           #C_E_Q_Unit := #C_E_Q_Unit + 1;
       ELSIF ((#E_Reactive_Rate1_Import < #MIN_ENERGY_VALUE) AND (#E_Reactive_Rate2_Import < #MIN_ENERGY_VALUE) AND
           (#E_Reactive_Rate1_Export < #MIN_ENERGY_VALUE) AND (#E_Reactive_Rate2_Export < #MIN_ENERGY_VALUE))
           AND (#C_E_Q_Unit > 1) THEN
           #C_E_Q_Unit := #C_E_Q_Unit - 1;
       ELSE
           ;
       END_IF;
       // selection apparent energy unit
       IF ((#E_Apparent_Rate1_Import > #MAX_ENERGY_VALUE) OR (#E_Apparent_Rate2_Import > #MAX_ENERGY_VALUE))
           AND (#C_E_S_Unit < 4) THEN
           #C_E_S_Unit := #C_E_S_Unit + 1;
       ELSIF ((#E_Apparent_Rate1_Import < #MIN_ENERGY_VALUE) AND (#E_Apparent_Rate2_Import < #MIN_ENERGY_VALUE))
           AND (#C_E_S_Unit > 1) THEN
           #C_E_S_Unit := #C_E_S_Unit - 1;
       ELSE
           ;
       END_IF;
   ELSE
       ;
   END_IF;
   //======================================================================================================================
   //==========calculate units=============================================================================================
   //======================================================================================================================    
   // calculate voltage unit
   CASE #C_U_Unit OF
       1:
           #U_Unit := 'mV';
           #U_L1_L2 := #ZU_L1_L2 * #THOUSAND;
           #U_L2_L3 := #ZU_L2_L3 * #THOUSAND;
           #U_L3_L1 := #ZU_L3_L1 * #THOUSAND;
           #U_L1 := #ZU_L1 * #THOUSAND;
           #U_L2 := #ZU_L2 * #THOUSAND;
           #U_L3 := #ZU_L3 * #THOUSAND;
           #U_L1_L2_min := #ZU_L1_L2_min * #THOUSAND;
           #U_L2_L3_min := #ZU_L2_L3_min * #THOUSAND;
           #U_L3_L1_min := #ZU_L3_L1_min * #THOUSAND;
           #U_L1_min := #ZU_L1_min * #THOUSAND;
           #U_L2_min := #ZU_L2_min * #THOUSAND;
           #U_L3_min := #ZU_L3_min * #THOUSAND;
           #U_L1_L2_max := #ZU_L1_L2_max * #THOUSAND;
           #U_L2_L3_max := #ZU_L2_L3_max * #THOUSAND;
           #U_L3_L1_max := #ZU_L3_L1_max * #THOUSAND;
           #U_L1_max := #ZU_L1_max * #THOUSAND;
           #U_L2_max := #ZU_L2_max * #THOUSAND;
           #U_L3_max := #ZU_L3_max * #THOUSAND;
           #U_PH_PH_Average := #ZU_PH_PH_Average * #THOUSAND;
           #U_PH_N_Average := #ZU_PH_N_Average * #THOUSAND;
           #U_PH_PH_Average_min := #ZU_PH_PH_Average_min * #THOUSAND;
           #U_PH_N_Average_min := #ZU_PH_N_Average_min * #THOUSAND;
           #U_PH_PH_Average_max := #ZU_PH_PH_Average_max * #THOUSAND;
           #U_PH_N_Average_max := #ZU_PH_N_Average_max * #THOUSAND;
       2:
           #U_Unit := 'V';
           #U_L1_L2 := #ZU_L1_L2;
           #U_L2_L3 := #ZU_L2_L3;
           #U_L3_L1 := #ZU_L3_L1;
           #U_L1 := #ZU_L1;
           #U_L2 := #ZU_L2;
           #U_L3 := #ZU_L3;
           #U_L1_L2_min := #ZU_L1_L2_min;
           #U_L2_L3_min := #ZU_L2_L3_min;
           #U_L3_L1_min := #ZU_L3_L1_min;
           #U_L1_min := #ZU_L1_min;
           #U_L2_min := #ZU_L2_min;
           #U_L3_min := #ZU_L3_min;
           #U_L1_L2_max := #ZU_L1_L2_max;
           #U_L2_L3_max := #ZU_L2_L3_max;
           #U_L3_L1_max := #ZU_L3_L1_max;
           #U_L1_max := #ZU_L1_max;
           #U_L2_max := #ZU_L2_max;
           #U_L3_max := #ZU_L3_max;
           #U_PH_PH_Average := #ZU_PH_PH_Average;
           #U_PH_N_Average := #ZU_PH_N_Average;
           #U_PH_PH_Average_min := #ZU_PH_PH_Average_min;
           #U_PH_N_Average_min := #ZU_PH_N_Average_min;
           #U_PH_PH_Average_max := #ZU_PH_PH_Average_max;
           #U_PH_N_Average_max := #ZU_PH_N_Average_max;
       ELSE:
           #U_Unit := 'kV';
           #U_L1_L2 := #ZU_L1_L2 / #THOUSAND;
           #U_L2_L3 := #ZU_L2_L3 / #THOUSAND;
           #U_L3_L1 := #ZU_L3_L1 / #THOUSAND;
           #U_L1 := #ZU_L1 / #THOUSAND;
           #U_L2 := #ZU_L2 / #THOUSAND;
           #U_L3 := #ZU_L3 / #THOUSAND;
           #U_L1_L2_min := #ZU_L1_L2_min / #THOUSAND;
           #U_L2_L3_min := #ZU_L2_L3_min / #THOUSAND;
           #U_L3_L1_min := #ZU_L3_L1_min / #THOUSAND;
           #U_L1_min := #ZU_L1_min / #THOUSAND;
           #U_L2_min := #ZU_L2_min / #THOUSAND;
           #U_L3_min := #ZU_L3_min / #THOUSAND;
           #U_L1_L2_max := #ZU_L1_L2_max / #THOUSAND;
           #U_L2_L3_max := #ZU_L2_L3_max / #THOUSAND;
           #U_L3_L1_max := #ZU_L3_L1_max / #THOUSAND;
           #U_L1_max := #ZU_L1_max / #THOUSAND;
           #U_L2_max := #ZU_L2_max / #THOUSAND;
           #U_L3_max := #ZU_L3_max / #THOUSAND;
           #U_PH_PH_Average := #ZU_PH_PH_Average / #THOUSAND;
           #U_PH_N_Average := #ZU_PH_N_Average / #THOUSAND;
           #U_PH_PH_Average_min := #ZU_PH_PH_Average_min / #THOUSAND;
           #U_PH_N_Average_min := #ZU_PH_N_Average_min / #THOUSAND;
           #U_PH_PH_Average_max := #ZU_PH_PH_Average_max / #THOUSAND;
           #U_PH_N_Average_max := #ZU_PH_N_Average_max / #THOUSAND;
   END_CASE;
   // calculate current unit    
   CASE #C_I_Unit OF
       1:
           #I_Unit := 'mA';
           #I_L1 := #ZI_L1 * #THOUSAND;
           #I_L2 := #ZI_L2 * #THOUSAND;
           #I_L3 := #ZI_L3 * #THOUSAND;
           #I_L1_min := #ZI_L1_min * #THOUSAND;
           #I_L2_min := #ZI_L2_min * #THOUSAND;
           #I_L3_min := #ZI_L3_min * #THOUSAND;
           #I_L1_max := #ZI_L1_max * #THOUSAND;
           #I_L2_max := #ZI_L2_max * #THOUSAND;
           #I_L3_max := #ZI_L3_max * #THOUSAND;
           #I_Average := #ZI_Average * #THOUSAND;
           #I_Average_min := #ZI_Average_min * #THOUSAND;
           #I_Average_max := #ZI_Average_max * #THOUSAND;
       2:
           #I_Unit := 'A';
           #I_L1 := #ZI_L1;
           #I_L2 := #ZI_L2;
           #I_L3 := #ZI_L3;
           #I_L1_min := #ZI_L1_min;
           #I_L2_min := #ZI_L2_min;
           #I_L3_min := #ZI_L3_min;
           #I_L1_max := #ZI_L1_max;
           #I_L2_max := #ZI_L2_max;
           #I_L3_max := #ZI_L3_max;
           #I_Average := #ZI_Average;
           #I_Average_min := #ZI_Average_min;
           #I_Average_max := #ZI_Average_max;
       ELSE:
           #I_Unit := 'kA';
           #I_L1 := #ZI_L1 / #THOUSAND;
           #I_L2 := #ZI_L2 / #THOUSAND;
           #I_L3 := #ZI_L3 / #THOUSAND;
           #I_L1_min := #ZI_L1_min / #THOUSAND;
           #I_L2_min := #ZI_L2_min / #THOUSAND;
           #I_L3_min := #ZI_L3_min / #THOUSAND;
           #I_L1_max := #ZI_L1_max / #THOUSAND;
           #I_L2_max := #ZI_L2_max / #THOUSAND;
           #I_L3_max := #ZI_L3_max / #THOUSAND;
           #I_Average := #ZI_Average / #THOUSAND;
           #I_Average_min := #ZI_Average_min / #THOUSAND;
           #I_Average_max := #ZI_Average_max / #THOUSAND;
   END_CASE;
   // calculate apparent power unit
   CASE #C_S_Unit OF
       1:
           #S_Unit := 'VA';
           #S_Total := #ZS_Total;
           #S_Total_min := #ZS_Total_min;
           #S_Total_max := #ZS_Total_max;
           #S_L1 := #ZS_L1;
           #S_L2 := #ZS_L2;
           #S_L3 := #ZS_L3;
           #S_L1_min := #ZS_L1_min;
           #S_L2_min := #ZS_L2_min;
           #S_L3_min := #ZS_L3_min;
           #S_L1_max := #ZS_L1_max;
           #S_L2_max := #ZS_L2_max;
           #S_L3_max := #ZS_L3_max;
       2:
           #S_Unit := 'kVA';
           #S_Total := #ZS_Total / #THOUSAND;
           #S_Total_min := #ZS_Total_min / #THOUSAND;
           #S_Total_max := #ZS_Total_max / #THOUSAND;
           #S_L1 := #ZS_L1 / #THOUSAND;
           #S_L2 := #ZS_L2 / #THOUSAND;
           #S_L3 := #ZS_L3 / #THOUSAND;
           #S_L1_min := #ZS_L1_min / #THOUSAND;
           #S_L2_min := #ZS_L2_min / #THOUSAND;
           #S_L3_min := #ZS_L3_min / #THOUSAND;
           #S_L1_max := #ZS_L1_max / #THOUSAND;
           #S_L2_max := #ZS_L2_max / #THOUSAND;
           #S_L3_max := #ZS_L3_max / #THOUSAND;
       3:
           #S_Unit := 'MVA';
           #S_Total := #ZS_Total / #MILLION;
           #S_Total_min := #ZS_Total_min / #MILLION;
           #S_Total_max := #ZS_Total_max / #MILLION;
           #S_L1 := #ZS_L1 / #MILLION;
           #S_L2 := #ZS_L2 / #MILLION;
           #S_L3 := #ZS_L3 / #MILLION;
           #S_L1_min := #ZS_L1_min / #MILLION;
           #S_L2_min := #ZS_L2_min / #MILLION;
           #S_L3_min := #ZS_L3_min / #MILLION;
           #S_L1_max := #ZS_L1_max / #MILLION;
           #S_L2_max := #ZS_L2_max / #MILLION;
           #S_L3_max := #ZS_L3_max / #MILLION;
       ELSE:
           #S_Unit := 'GVA';
           #S_Total := #ZS_Total / #MILLION / #THOUSAND;
           #S_Total_min := #ZS_Total_min / #MILLION / #THOUSAND;
           #S_Total_max := #ZS_Total_max / #MILLION / #THOUSAND;
           #S_L1 := #ZS_L1 / #MILLION / #THOUSAND;
           #S_L2 := #ZS_L2 / #MILLION / #THOUSAND;
           #S_L3 := #ZS_L3 / #MILLION / #THOUSAND;
           #S_L1_min := #ZS_L1_min / #MILLION / #THOUSAND;
           #S_L2_min := #ZS_L2_min / #MILLION / #THOUSAND;
           #S_L3_min := #ZS_L3_min / #MILLION / #THOUSAND;
           #S_L1_max := #ZS_L1_max / #MILLION / #THOUSAND;
           #S_L2_max := #ZS_L2_max / #MILLION / #THOUSAND;
           #S_L3_max := #ZS_L3_max / #MILLION / #THOUSAND;
   END_CASE;
   // calculate active power unit    
   CASE #C_P_Unit OF
       1:
           #P_Unit := 'W';
           #P_Total := #ZP_Total;
           #P_Total_min := #ZP_Total_min;
           #P_Total_max := #ZP_Total_max;
           #P_L1 := #ZP_L1;
           #P_L2 := #ZP_L2;
           #P_L3 := #ZP_L3;
           #P_L1_min := #ZP_L1_min;
           #P_L2_min := #ZP_L2_min;
           #P_L3_min := #ZP_L3_min;
           #P_L1_max := #ZP_L1_max;
           #P_L2_max := #ZP_L2_max;
           #P_L3_max := #ZP_L3_max;
       2:
           #P_Unit := 'kW';
           #P_Total := #ZP_Total / #THOUSAND;
           #P_Total_min := #ZP_Total_min / #THOUSAND;
           #P_Total_max := #ZP_Total_max / #THOUSAND;
           #P_L1 := #ZP_L1 / #THOUSAND;
           #P_L2 := #ZP_L2 / #THOUSAND;
           #P_L3 := #ZP_L3 / #THOUSAND;
           #P_L1_min := #ZP_L1_min / #THOUSAND;
           #P_L2_min := #ZP_L2_min / #THOUSAND;
           #P_L3_min := #ZP_L3_min / #THOUSAND;
           #P_L1_max := #ZP_L1_max / #THOUSAND;
           #P_L2_max := #ZP_L2_max / #THOUSAND;
           #P_L3_max := #ZP_L3_max / #THOUSAND;
       3:
           #P_Unit := 'MW';
           #P_Total := #ZP_Total / #MILLION;
           #P_Total_min := #ZP_Total_min / #MILLION;
           #P_Total_max := #ZP_Total_max / #MILLION;
           #P_L1 := #ZP_L1 / #MILLION;
           #P_L2 := #ZP_L2 / #MILLION;
           #P_L3 := #ZP_L3 / #MILLION;
           #P_L1_min := #ZP_L1_min / #MILLION;
           #P_L2_min := #ZP_L2_min / #MILLION;
           #P_L3_min := #ZP_L3_min / #MILLION;
           #P_L1_max := #ZP_L1_max / #MILLION;
           #P_L2_max := #ZP_L2_max / #MILLION;
           #P_L3_max := #ZP_L3_max / #MILLION;
       ELSE:
           #P_Unit := 'GW';
           #P_Total := #ZP_Total / #MILLION / #THOUSAND;
           #P_Total_min := #ZP_Total_min / #MILLION / #THOUSAND;
           #P_Total_max := #ZP_Total_max / #MILLION / #THOUSAND;
           #P_L1 := #ZP_L1 / #MILLION / #THOUSAND;
           #P_L2 := #ZP_L2 / #MILLION / #THOUSAND;
           #P_L3 := #ZP_L3 / #MILLION / #THOUSAND;
           #P_L1_min := #ZP_L1_min / #MILLION / #THOUSAND;
           #P_L2_min := #ZP_L2_min / #MILLION / #THOUSAND;
           #P_L3_min := #ZP_L3_min / #MILLION / #THOUSAND;
           #P_L1_max := #ZP_L1_max / #MILLION / #THOUSAND;
           #P_L2_max := #ZP_L2_max / #MILLION / #THOUSAND;
           #P_L3_max := #ZP_L3_max / #MILLION / #THOUSAND;
   END_CASE;
   // calculate reactive power unit   
   CASE #C_Q_Unit OF
       1:
           #Q_Unit := 'var';
           #Q_Total := #ZQ_Total;
           #Q_Total_min := #ZQ_Total_min;
           #Q_Total_max := #ZQ_Total_max;
           #Q_L1 := #ZQ_L1;
           #Q_L2 := #ZQ_L2;
           #Q_L3 := #ZQ_L3;
           #Q_L1_min := #ZQ_L1_min;
           #Q_L2_min := #ZQ_L2_min;
           #Q_L3_min := #ZQ_L3_min;
           #Q_L1_max := #ZQ_L1_max;
           #Q_L2_max := #ZQ_L2_max;
           #Q_L3_max := #ZQ_L3_max;
       2:
           #Q_Unit := 'kvar';
           #Q_Total := #ZQ_Total / #THOUSAND;
           #Q_Total_min := #ZQ_Total_min / #THOUSAND;
           #Q_Total_max := #ZQ_Total_max / #THOUSAND;
           #Q_L1 := #ZQ_L1 / #THOUSAND;
           #Q_L2 := #ZQ_L2 / #THOUSAND;
           #Q_L3 := #ZQ_L3 / #THOUSAND;
           #Q_L1_min := #ZQ_L1_min / #THOUSAND;
           #Q_L2_min := #ZQ_L2_min / #THOUSAND;
           #Q_L3_min := #ZQ_L3_min / #THOUSAND;
           #Q_L1_max := #ZQ_L1_max / #THOUSAND;
           #Q_L2_max := #ZQ_L2_max / #THOUSAND;
           #Q_L3_max := #ZQ_L3_max / #THOUSAND;
       3:
           #Q_Unit := 'Mvar';
           #Q_Total := #ZQ_Total / #MILLION;
           #Q_Total_min := #ZQ_Total_min / #MILLION;
           #Q_Total_max := #ZQ_Total_max / #MILLION;
           #Q_L1 := #ZQ_L1 / #MILLION;
           #Q_L2 := #ZQ_L2 / #MILLION;
           #Q_L3 := #ZQ_L3 / #MILLION;
           #Q_L1_min := #ZQ_L1_min / #MILLION;
           #Q_L2_min := #ZQ_L2_min / #MILLION;
           #Q_L3_min := #ZQ_L3_min / #MILLION;
           #Q_L1_max := #ZQ_L1_max / #MILLION;
           #Q_L2_max := #ZQ_L2_max / #MILLION;
           #Q_L3_max := #ZQ_L3_max / #MILLION;
       ELSE:
           #Q_Unit := 'Gvar';
           #Q_Total := #ZQ_Total / #MILLION / #THOUSAND;
           #Q_Total_min := #ZQ_Total_min / #MILLION / #THOUSAND;
           #Q_Total_max := #ZQ_Total_max / #MILLION / #THOUSAND;
           #Q_L1 := #ZQ_L1 / #MILLION / #THOUSAND;
           #Q_L2 := #ZQ_L2 / #MILLION / #THOUSAND;
           #Q_L3 := #ZQ_L3 / #MILLION / #THOUSAND;
           #Q_L1_min := #ZQ_L1_min / #MILLION / #THOUSAND;
           #Q_L2_min := #ZQ_L2_min / #MILLION / #THOUSAND;
           #Q_L3_min := #ZQ_L3_min / #MILLION / #THOUSAND;
           #Q_L1_max := #ZQ_L1_max / #MILLION / #THOUSAND;
           #Q_L2_max := #ZQ_L2_max / #MILLION / #THOUSAND;
           #Q_L3_max := #ZQ_L3_max / #MILLION / #THOUSAND;
   END_CASE;
   // calculate apparent energy unit     
   CASE #C_E_S_Unit OF
       1:
           IF ((#VEnergy_Meter_Unit[9] = TRUE) OR (#VEnergy_Meter_Unit[10] = TRUE)) THEN
               #S_Energy_Unit := 'kVAh';
               IF (#VEnergy_Meter_Unit[9] = FALSE) THEN
                   #E_Apparent_Rate1_Import := #ZE_Apparent_Rate1_Import / #THOUSAND;
               ELSE
                   #E_Apparent_Rate1_Import := #ZE_Apparent_Rate1_Import;
               END_IF;
               IF (#VEnergy_Meter_Unit[10] = FALSE) THEN
                   #E_Apparent_Rate2_Import := #ZE_Apparent_Rate2_Import / #THOUSAND;
               ELSE
                   #E_Apparent_Rate2_Import := #ZE_Apparent_Rate2_Import;
               END_IF;
           ELSE
               #S_Energy_Unit := 'VAh';
               #E_Apparent_Rate1_Import := #ZE_Apparent_Rate1_Import;
               #E_Apparent_Rate2_Import := #ZE_Apparent_Rate2_Import;
           END_IF;
       2:
           IF ((#VEnergy_Meter_Unit[9] = TRUE) OR (#VEnergy_Meter_Unit[10] = TRUE)) THEN
               #S_Energy_Unit := 'MVAh';
               IF (#VEnergy_Meter_Unit[9] = FALSE) THEN
                   #E_Apparent_Rate1_Import := #ZE_Apparent_Rate1_Import / #MILLION;
               ELSE
                   #E_Apparent_Rate1_Import := #ZE_Apparent_Rate1_Import / #THOUSAND;
               END_IF;
               IF (#VEnergy_Meter_Unit[10] = FALSE) THEN
                   #E_Apparent_Rate2_Import := #ZE_Apparent_Rate2_Import / #MILLION;
               ELSE
                   #E_Apparent_Rate2_Import := #ZE_Apparent_Rate2_Import / #THOUSAND;
               END_IF;
           ELSE
               #S_Energy_Unit := 'kVAh';
               #E_Apparent_Rate1_Import := #ZE_Apparent_Rate1_Import / #THOUSAND;
               #E_Apparent_Rate2_Import := #ZE_Apparent_Rate2_Import / #THOUSAND;
           END_IF;
       3:
           IF ((#VEnergy_Meter_Unit[9] = TRUE) OR (#VEnergy_Meter_Unit[10] = TRUE)) THEN
               #S_Energy_Unit := 'GVAh';
               IF (#VEnergy_Meter_Unit[9] = FALSE) THEN
                   #E_Apparent_Rate1_Import := #ZE_Apparent_Rate1_Import / #MILLION / #THOUSAND;
               ELSE
                   #E_Apparent_Rate1_Import := #ZE_Apparent_Rate1_Import / #MILLION;
               END_IF;
               IF (#VEnergy_Meter_Unit[10] = FALSE) THEN
                   #E_Apparent_Rate2_Import := #ZE_Apparent_Rate2_Import / #MILLION / #THOUSAND;
               ELSE
                   #E_Apparent_Rate2_Import := #ZE_Apparent_Rate2_Import / #MILLION;
               END_IF;
           ELSE
               #S_Energy_Unit := 'MVAh';
               #E_Apparent_Rate1_Import := #ZE_Apparent_Rate1_Import / #MILLION;
               #E_Apparent_Rate2_Import := #ZE_Apparent_Rate2_Import / #MILLION;
           END_IF;
       ELSE:
           IF ((#VEnergy_Meter_Unit[9] = TRUE) OR (#VEnergy_Meter_Unit[10] = TRUE)) THEN
               #S_Energy_Unit := 'TVAh';
               IF (#VEnergy_Meter_Unit[9] = FALSE) THEN
                   #E_Apparent_Rate1_Import := #ZE_Apparent_Rate1_Import / #MILLION / #MILLION;
               ELSE
                   #E_Apparent_Rate1_Import := #ZE_Apparent_Rate1_Import / #MILLION / #THOUSAND;
               END_IF;
               IF (#VEnergy_Meter_Unit[10] = FALSE) THEN
                   #E_Apparent_Rate2_Import := #ZE_Apparent_Rate2_Import / #MILLION / #MILLION;
               ELSE
                   #E_Apparent_Rate2_Import := #ZE_Apparent_Rate2_Import / #MILLION / #THOUSAND;
               END_IF;
           ELSE
               #S_Energy_Unit := 'GVAh';
               #E_Apparent_Rate1_Import := #ZE_Apparent_Rate1_Import / #MILLION / #THOUSAND;
               #E_Apparent_Rate2_Import := #ZE_Apparent_Rate2_Import / #MILLION / #THOUSAND;
           END_IF;
   END_CASE;
   // calculate active energy unit     
   CASE #C_E_P_Unit OF
       1:
           IF ((#VEnergy_Meter_Unit[1] = TRUE) OR (#VEnergy_Meter_Unit[2] = TRUE) OR
               (#VEnergy_Meter_Unit[3] = TRUE) OR (#VEnergy_Meter_Unit[4] = TRUE)) THEN
               #P_Energy_Unit := 'kWh';
               IF (#VEnergy_Meter_Unit[1] = FALSE) THEN
                   #E_Active_Rate1_Import := #ZE_Active_Rate1_Import / #THOUSAND;
               ELSE
                   #E_Active_Rate1_Import := #ZE_Active_Rate1_Import;
               END_IF;
               IF (#VEnergy_Meter_Unit[2] = FALSE) THEN
                   #E_Active_Rate2_Import := #ZE_Active_Rate2_Import / #THOUSAND;
               ELSE
                   #E_Active_Rate2_Import := #ZE_Active_Rate2_Import;
               END_IF;
               IF (#VEnergy_Meter_Unit[3] = FALSE) THEN
                   #E_Active_Rate1_Export := #ZE_Active_Rate1_Export / #THOUSAND;
               ELSE
                   #E_Active_Rate1_Export := #ZE_Active_Rate1_Export;
               END_IF;
               IF (#VEnergy_Meter_Unit[4] = FALSE) THEN
                   #E_Active_Rate1_Export := #ZE_Active_Rate1_Export / #THOUSAND;
               ELSE
                   #E_Active_Rate1_Export := #ZE_Active_Rate1_Export;
               END_IF;
           ELSE
               #P_Energy_Unit := 'Wh';
               #E_Active_Rate1_Import := #ZE_Active_Rate1_Import;
               #E_Active_Rate2_Import := #ZE_Active_Rate2_Import;
               #E_Active_Rate1_Export := #ZE_Active_Rate1_Export;
               #E_Active_Rate2_Export := #ZE_Active_Rate2_Export;
           END_IF;
       2:
           IF ((#VEnergy_Meter_Unit[1] = TRUE) OR (#VEnergy_Meter_Unit[2] = TRUE) OR
               (#VEnergy_Meter_Unit[3] = TRUE) OR (#VEnergy_Meter_Unit[4] = TRUE)) THEN
               #P_Energy_Unit := 'MWh';
               IF (#VEnergy_Meter_Unit[1] = FALSE) THEN
                   #E_Active_Rate1_Import := #ZE_Active_Rate1_Import / #MILLION;
               ELSE
                   #E_Active_Rate1_Import := #ZE_Active_Rate1_Import / #THOUSAND;
               END_IF;
               IF (#VEnergy_Meter_Unit[2] = FALSE) THEN
                   #E_Active_Rate2_Import := #ZE_Active_Rate2_Import / #MILLION;
               ELSE
                   #E_Active_Rate2_Import := #ZE_Active_Rate2_Import / #THOUSAND;
               END_IF;
               IF (#VEnergy_Meter_Unit[3] = FALSE) THEN
                   #E_Active_Rate1_Export := #ZE_Active_Rate1_Export / #MILLION;
               ELSE
                   #E_Active_Rate1_Export := #ZE_Active_Rate1_Export / #THOUSAND;
               END_IF;
               IF (#VEnergy_Meter_Unit[4] = FALSE) THEN
                   #E_Active_Rate2_Export := #ZE_Active_Rate2_Export / #MILLION;
               ELSE
                   #E_Active_Rate2_Export := #ZE_Active_Rate2_Export / #THOUSAND;
               END_IF;
           ELSE
               #P_Energy_Unit := 'kWh';
               #E_Active_Rate1_Import := #ZE_Active_Rate1_Import / #THOUSAND;
               #E_Active_Rate2_Import := #ZE_Active_Rate2_Import / #THOUSAND;
               #E_Active_Rate1_Export := #ZE_Active_Rate1_Export / #THOUSAND;
               #E_Active_Rate2_Export := #ZE_Active_Rate2_Export / #THOUSAND;
           END_IF;
       3:
           IF ((#VEnergy_Meter_Unit[1] = TRUE) OR (#VEnergy_Meter_Unit[2] = TRUE) OR
               (#VEnergy_Meter_Unit[3] = TRUE) OR (#VEnergy_Meter_Unit[4] = TRUE)) THEN
               #P_Energy_Unit := 'GWh';
               IF (#VEnergy_Meter_Unit[1] = FALSE) THEN
                   #E_Active_Rate1_Import := #ZE_Active_Rate1_Import / #MILLION / #THOUSAND;
               ELSE
                   #E_Active_Rate1_Import := #ZE_Active_Rate1_Import / #MILLION;
               END_IF;
               IF (#VEnergy_Meter_Unit[2] = FALSE) THEN
                   #E_Active_Rate2_Import := #ZE_Active_Rate2_Import / #MILLION / #THOUSAND;
               ELSE
                   #E_Active_Rate2_Import := #ZE_Active_Rate2_Import / #MILLION;
               END_IF;
               IF (#VEnergy_Meter_Unit[3] = FALSE) THEN
                   #E_Active_Rate1_Export := #ZE_Active_Rate1_Export / #MILLION / #THOUSAND;
               ELSE
                   #E_Active_Rate1_Export := #ZE_Active_Rate1_Export / #MILLION;
               END_IF;
               IF (#VEnergy_Meter_Unit[4] = FALSE) THEN
                   #E_Active_Rate2_Export := #ZE_Active_Rate2_Export / #MILLION / #THOUSAND;
               ELSE
                   #E_Active_Rate2_Export := #ZE_Active_Rate2_Export / #MILLION;
               END_IF;
           ELSE
               #P_Energy_Unit := 'MWh';
               #E_Active_Rate1_Import := #ZE_Active_Rate1_Import / #MILLION;
               #E_Active_Rate2_Import := #ZE_Active_Rate2_Import / #MILLION;
               #E_Active_Rate1_Export := #ZE_Active_Rate1_Export / #MILLION;
               #E_Active_Rate2_Export := #ZE_Active_Rate2_Export / #MILLION;
           END_IF;
       ELSE:
           IF ((#VEnergy_Meter_Unit[1] = TRUE) OR (#VEnergy_Meter_Unit[2] = TRUE) OR
               (#VEnergy_Meter_Unit[3] = TRUE) OR (#VEnergy_Meter_Unit[4] = TRUE)) THEN
               #P_Energy_Unit := 'TWh';
               IF (#VEnergy_Meter_Unit[1] = FALSE) THEN
                   #E_Active_Rate1_Import := #ZE_Active_Rate1_Import / #MILLION / #MILLION;
               ELSE
                   #E_Active_Rate1_Import := #ZE_Active_Rate1_Import / #MILLION / #THOUSAND;
               END_IF;
               IF (#VEnergy_Meter_Unit[2] = FALSE) THEN
                   #E_Active_Rate2_Import := #ZE_Active_Rate2_Import / #MILLION / #MILLION;
               ELSE
                   #E_Active_Rate2_Import := #ZE_Active_Rate2_Import / #MILLION / #THOUSAND;
               END_IF;
               IF (#VEnergy_Meter_Unit[3] = FALSE) THEN
                   #E_Active_Rate1_Export := #ZE_Active_Rate1_Export / #MILLION / #MILLION;
               ELSE
                   #E_Active_Rate1_Export := #ZE_Active_Rate1_Export / #MILLION / #THOUSAND;
               END_IF;
               IF (#VEnergy_Meter_Unit[4] = FALSE) THEN
                   #E_Active_Rate2_Export := #ZE_Active_Rate2_Export / #MILLION / #MILLION;
               ELSE
                   #E_Active_Rate2_Export := #ZE_Active_Rate2_Export / #MILLION / #THOUSAND;
               END_IF;
           ELSE
               #P_Energy_Unit := 'GWh';
               #E_Active_Rate1_Import := #ZE_Active_Rate1_Import / #MILLION / #THOUSAND;
               #E_Active_Rate2_Import := #ZE_Active_Rate2_Import / #MILLION / #THOUSAND;
               #E_Active_Rate1_Export := #ZE_Active_Rate1_Export / #MILLION / #THOUSAND;
               #E_Active_Rate2_Export := #ZE_Active_Rate2_Export / #MILLION / #THOUSAND;
           END_IF;
   END_CASE;
   // calculate reactive energy unit     
   CASE #C_E_Q_Unit OF
       1:
           IF ((#VEnergy_Meter_Unit[5] = TRUE) OR (#VEnergy_Meter_Unit[6] = TRUE) OR
               (#VEnergy_Meter_Unit[7] = TRUE) OR (#VEnergy_Meter_Unit[8] = TRUE)) THEN
               #Q_Energy_Unit := 'kWh';
               IF (#VEnergy_Meter_Unit[5] = FALSE) THEN
                   #E_Reactive_Rate1_Import := #ZE_Reactive_Rate1_Import / #THOUSAND;
               ELSE
                   #E_Reactive_Rate1_Import := #ZE_Reactive_Rate1_Import;
               END_IF;
               IF (#VEnergy_Meter_Unit[6] = FALSE) THEN
                   #E_Reactive_Rate2_Import := #ZE_Reactive_Rate2_Import / #THOUSAND;
               ELSE
                   #E_Reactive_Rate2_Import := #ZE_Reactive_Rate2_Import;
               END_IF;
               IF (#VEnergy_Meter_Unit[7] = FALSE) THEN
                   #E_Reactive_Rate1_Export := #ZE_Reactive_Rate1_Export / #THOUSAND;
               ELSE
                   #E_Reactive_Rate1_Export := #ZE_Reactive_Rate1_Export;
               END_IF;
               IF (#VEnergy_Meter_Unit[8] = FALSE) THEN
                   #E_Reactive_Rate2_Export := #ZE_Reactive_Rate2_Export / #THOUSAND;
               ELSE
                   #E_Reactive_Rate2_Export := #ZE_Reactive_Rate2_Export;
               END_IF;
           ELSE
               #Q_Energy_Unit := 'varh';
               #E_Reactive_Rate1_Import := #ZE_Reactive_Rate1_Import;
               #E_Reactive_Rate2_Import := #ZE_Reactive_Rate2_Import;
               #E_Reactive_Rate1_Export := #ZE_Reactive_Rate1_Export;
               #E_Reactive_Rate2_Export := #ZE_Reactive_Rate2_Export;
           END_IF;
       2:
           IF ((#VEnergy_Meter_Unit[5] = TRUE) OR (#VEnergy_Meter_Unit[6] = TRUE) OR
               (#VEnergy_Meter_Unit[7] = TRUE) OR (#VEnergy_Meter_Unit[8] = TRUE)) THEN
               #Q_Energy_Unit := 'MWh';
               IF (#VEnergy_Meter_Unit[5] = FALSE) THEN
                   #E_Reactive_Rate1_Import := #ZE_Reactive_Rate1_Import / #MILLION;
               ELSE
                   #E_Reactive_Rate1_Import := #ZE_Reactive_Rate1_Import;
               END_IF;
               IF (#VEnergy_Meter_Unit[6] = FALSE) THEN
                   #E_Reactive_Rate2_Import := #ZE_Reactive_Rate2_Import / #MILLION;
               ELSE
                   #E_Reactive_Rate2_Import := #ZE_Reactive_Rate2_Import;
               END_IF;
               IF (#VEnergy_Meter_Unit[7] = FALSE) THEN
                   #E_Reactive_Rate1_Export := #ZE_Reactive_Rate1_Export / #MILLION;
               ELSE
                   #E_Reactive_Rate1_Export := #ZE_Reactive_Rate1_Export;
               END_IF;
               IF (#VEnergy_Meter_Unit[8] = FALSE) THEN
                   #E_Reactive_Rate2_Export := #ZE_Reactive_Rate2_Export / #MILLION;
               ELSE
                   #E_Reactive_Rate2_Export := #ZE_Reactive_Rate2_Export;
               END_IF;
           ELSE
               #Q_Energy_Unit := 'kvarh';
               #E_Reactive_Rate1_Import := #ZE_Reactive_Rate1_Import / #THOUSAND;
               #E_Reactive_Rate2_Import := #ZE_Reactive_Rate2_Import / #THOUSAND;
               #E_Reactive_Rate1_Export := #ZE_Reactive_Rate1_Export / #THOUSAND;
               #E_Reactive_Rate2_Export := #ZE_Reactive_Rate2_Export / #THOUSAND;
           END_IF;
       3:
           IF ((#VEnergy_Meter_Unit[5] = TRUE) OR (#VEnergy_Meter_Unit[6] = TRUE) OR
               (#VEnergy_Meter_Unit[7] = TRUE) OR (#VEnergy_Meter_Unit[8] = TRUE)) THEN
               #Q_Energy_Unit := 'GWh';
               IF (#VEnergy_Meter_Unit[5] = FALSE) THEN
                   #E_Reactive_Rate1_Import := #ZE_Reactive_Rate1_Import / #MILLION / #THOUSAND;
               ELSE
                   #E_Reactive_Rate1_Import := #ZE_Reactive_Rate1_Import / #THOUSAND;
               END_IF;
               IF (#VEnergy_Meter_Unit[6] = FALSE) THEN
                   #E_Reactive_Rate2_Import := #ZE_Reactive_Rate2_Import / #MILLION / #THOUSAND;
               ELSE
                   #E_Reactive_Rate2_Import := #ZE_Reactive_Rate2_Import / #THOUSAND;
               END_IF;
               IF (#VEnergy_Meter_Unit[7] = FALSE) THEN
                   #E_Reactive_Rate1_Export := #ZE_Reactive_Rate1_Export / #MILLION / #THOUSAND;
               ELSE
                   #E_Reactive_Rate1_Export := #ZE_Reactive_Rate1_Export / #THOUSAND;
               END_IF;
               IF (#VEnergy_Meter_Unit[8] = FALSE) THEN
                   #E_Reactive_Rate2_Export := #ZE_Reactive_Rate2_Export / #MILLION / #THOUSAND;
               ELSE
                   #E_Reactive_Rate2_Export := #ZE_Reactive_Rate2_Export / #THOUSAND;
               END_IF;
           ELSE
               #Q_Energy_Unit := 'Mvarh';
               #E_Reactive_Rate1_Import := #ZE_Reactive_Rate1_Import / #MILLION;
               #E_Reactive_Rate2_Import := #ZE_Reactive_Rate2_Import / #MILLION;
               #E_Reactive_Rate1_Export := #ZE_Reactive_Rate1_Export / #MILLION;
               #E_Reactive_Rate2_Export := #ZE_Reactive_Rate2_Export / #MILLION;
           END_IF;
       ELSE:
           IF ((#VEnergy_Meter_Unit[5] = TRUE) OR (#VEnergy_Meter_Unit[6] = TRUE) OR
               (#VEnergy_Meter_Unit[7] = TRUE) OR (#VEnergy_Meter_Unit[8] = TRUE)) THEN
               #Q_Energy_Unit := 'TWh';
               IF (#VEnergy_Meter_Unit[5] = FALSE) THEN
                   #E_Reactive_Rate1_Import := #ZE_Reactive_Rate1_Import / #MILLION / #MILLION;
               ELSE
                   #E_Reactive_Rate1_Import := #ZE_Reactive_Rate1_Import / #MILLION / #THOUSAND;
               END_IF;
               IF (#VEnergy_Meter_Unit[6] = FALSE) THEN
                   #E_Reactive_Rate2_Import := #ZE_Reactive_Rate2_Import / #MILLION / #MILLION;
               ELSE
                   #E_Reactive_Rate2_Import := #ZE_Reactive_Rate2_Import / #MILLION / #THOUSAND;
               END_IF;
               IF (#VEnergy_Meter_Unit[7] = FALSE) THEN
                   #E_Reactive_Rate1_Export := #ZE_Reactive_Rate1_Export / #MILLION / #MILLION;
               ELSE
                   #E_Reactive_Rate1_Export := #ZE_Reactive_Rate1_Export / #MILLION / #THOUSAND;
               END_IF;
               IF (#VEnergy_Meter_Unit[8] = FALSE) THEN
                   #E_Reactive_Rate2_Export := #ZE_Reactive_Rate2_Export / #MILLION / #MILLION;
               ELSE
                   #E_Reactive_Rate2_Export := #ZE_Reactive_Rate2_Export / #MILLION / #THOUSAND;
               END_IF;
           ELSE
               #Q_Energy_Unit := 'Gvarh';
               #E_Reactive_Rate1_Import := #ZE_Reactive_Rate1_Import / #MILLION / #THOUSAND;
               #E_Reactive_Rate2_Import := #ZE_Reactive_Rate2_Import / #MILLION / #THOUSAND;
               #E_Reactive_Rate1_Export := #ZE_Reactive_Rate1_Export / #MILLION / #THOUSAND;
               #E_Reactive_Rate2_Export := #ZE_Reactive_Rate2_Export / #MILLION / #THOUSAND;
           END_IF;
   END_CASE;
   //======================================================================================================================
   //==========calculate scale final value=================================================================================
   //======================================================================================================================        
   // calculate scale final voltage PH-PH
   IF ((#AREA_TO_THOUSAND < #U_L1_L2_max) OR (#AREA_TO_THOUSAND < #U_L2_L3_max) OR (#AREA_TO_THOUSAND < #U_L3_L1_max)) THEN
       #ZScale_End_U_PH_PH := #ZSCALE_END_I4;
   ELSIF ((#AREA_TO_HUNDRED < #U_L1_L2_max) OR (#AREA_TO_HUNDRED < #U_L2_L3_max) OR (#AREA_TO_HUNDRED < #U_L3_L1_max)) THEN
       #ZScale_End_U_PH_PH := #ZSCALE_END_I3;
   ELSIF ((#AREA_TO_TEN < #U_L1_L2_max) OR (#AREA_TO_TEN < #U_L2_L3_max) OR (#AREA_TO_TEN < #U_L3_L1_max)) THEN
       #ZScale_End_U_PH_PH := #ZSCALE_END_I2;
   ELSIF ((0 <= #U_L1_L2_max) OR (0 <= #U_L2_L3_max) OR (0 <= #U_L3_L1_max)) THEN
       #ZScale_End_U_PH_PH := #ZSCALE_END_I1;
   ELSE
       ;
   END_IF;
   // selection maximum value
   #U_PH_PH := MAX(IN1 := #U_L1_L2_max, IN2 := #U_L2_L3_max, IN3 := #U_L3_L1_max, IN4 := 4.0);
   // 
   #Scale_End_U_PH_PH := (REAL_TO_DINT(#U_PH_PH * #FACTOR)) + (#ZScale_End_U_PH_PH - (REAL_TO_DINT(#U_PH_PH * #FACTOR) MOD #ZScale_End_U_PH_PH));
   // calculate scale final voltage PH-N
   IF ((#AREA_TO_THOUSAND < #U_L1_max) OR (#AREA_TO_THOUSAND < #U_L2_max) OR (#AREA_TO_THOUSAND < #U_L3_max)) THEN
       #ZScale_End_U_PH_N := #ZSCALE_END_I4;
   ELSIF ((#AREA_TO_HUNDRED < #U_L1_max) OR (#AREA_TO_HUNDRED < #U_L2_max) OR (#AREA_TO_HUNDRED < #U_L3_max)) THEN
       #ZScale_End_U_PH_N := #ZSCALE_END_I3;
   ELSIF ((#AREA_TO_TEN < #U_L1_max) OR (#AREA_TO_TEN < #U_L2_max) OR (#AREA_TO_TEN < #U_L3_max)) THEN
       #ZScale_End_U_PH_N := #ZSCALE_END_I2;
   ELSIF ((0 <= #U_L1_max) OR (0 <= #U_L2_max) OR (0 <= #U_L3_max)) THEN
       #ZScale_End_U_PH_N := #ZSCALE_END_I1;
   ELSE
       ;
   END_IF;
   // selection maximum value
   #U_PH_N := MAX(IN1 := #U_L1_max, IN2 := #U_L2_max, IN3 := #U_L3_max, IN4 := 4.0);
   // 
   #Scale_End_U_PH_N := (REAL_TO_DINT(#U_PH_N * #FACTOR)) + (#ZScale_End_U_PH_N - (REAL_TO_DINT(#U_PH_N * #FACTOR) MOD #ZScale_End_U_PH_N));
   // calculate scale final current
   IF ((#AREA_TO_THOUSAND < #I_L1_max) OR (#AREA_TO_THOUSAND < #I_L2_max) OR (#AREA_TO_THOUSAND < #I_L3_max)) THEN
       #ZScale_End_I := #ZSCALE_END_I4;
   ELSIF ((#AREA_TO_HUNDRED < #I_L1_max) OR (#AREA_TO_HUNDRED < #I_L2_max) OR (#AREA_TO_HUNDRED < #I_L3_max)) THEN
       #ZScale_End_I := #ZSCALE_END_I3;
   ELSIF ((#AREA_TO_TEN < #I_L1_max) OR (#AREA_TO_TEN < #I_L2_max) OR (#AREA_TO_TEN < #I_L3_max)) THEN
       #ZScale_End_I := #ZSCALE_END_I2;
   ELSIF ((0 <= #I_L1_max) OR (0 <= #I_L2_max) OR (0 <= #I_L3_max)) THEN
       #ZScale_End_I := #ZSCALE_END_I1;
   ELSE
       ;
   END_IF;
   // selection maximum value
   #I := MAX(IN1 := #I_L1_max, IN2 := #I_L2_max, IN3 := #I_L3_max, IN4 := 4.0);
   //
   #Scale_End_I := (REAL_TO_DINT(#I * #FACTOR)) + (#ZScale_End_I - (REAL_TO_DINT(#I * #FACTOR) MOD #ZScale_End_I));
   // calculate scale final apparent power    
   IF ((#AREA_TO_THOUSAND < #S_L1_max) OR (#AREA_TO_THOUSAND < #S_L2_max) OR
       (#AREA_TO_THOUSAND < #S_L3_max) OR (#AREA_TO_THOUSAND < #S_Total_max)) THEN
       #ZScale_End_S := #ZSCALE_END_SPQ4;
   ELSIF ((#AREA_TO_HUNDRED < #S_L1_max) OR (#AREA_TO_HUNDRED < #S_L2_max) OR
       (#AREA_TO_HUNDRED < #S_L3_max) OR (#AREA_TO_HUNDRED < #S_Total_max)) THEN
       #ZScale_End_S := #ZSCALE_END_SPQ3;
   ELSIF ((#AREA_TO_TEN < #S_L1_max) OR (#AREA_TO_TEN < #S_L2_max) OR
       (#AREA_TO_TEN < #S_L3_max) OR (#AREA_TO_TEN < #S_Total_max)) THEN
       #ZScale_End_S := #ZSCALE_END_SPQ2;
   ELSIF ((0 <= #S_L1_max) OR (0 <= #S_L2_max) OR (0 <= #S_L3_max) OR (0 <= #S_Total_max)) THEN
       #ZScale_End_S := #ZSCALE_END_SPQ1;
   ELSE
       ;
   END_IF;
   // selection maximum value 
   #S := MAX(IN1 := #S_L1_max, IN2 := #S_L2_max, IN3 := #S_L3_max, IN4 := #S_Total_max, IN5 := 4.0);
   //
   #Scale_End_S := (REAL_TO_DINT(#S * #FACTOR)) + (#ZScale_End_S - (REAL_TO_DINT(#S * #FACTOR) MOD #ZScale_End_S));
   // calculate scale final active power
   IF ((#AREA_TO_THOUSAND < #P_L1_max) OR (#AREA_TO_THOUSAND < #P_L2_max) OR
       (#AREA_TO_THOUSAND < #P_L3_max) OR (#AREA_TO_THOUSAND < #P_Total_max)) THEN
       #ZScale_End_P := #ZSCALE_END_SPQ4;
   ELSIF ((#AREA_TO_HUNDRED < #P_L1_max) OR (#AREA_TO_HUNDRED < #P_L2_max) OR
       (#AREA_TO_HUNDRED < #P_L3_max) OR (#AREA_TO_HUNDRED < #P_Total_max)) THEN
       #ZScale_End_P := #ZSCALE_END_SPQ3;
   ELSIF ((#AREA_TO_TEN < #P_L1_max) OR (#AREA_TO_TEN < #P_L2_max) OR
       (#AREA_TO_TEN < #P_L3_max) OR (#AREA_TO_TEN < #P_Total_max)) THEN
       #ZScale_End_P := #ZSCALE_END_SPQ2;
   ELSIF ((0 <= #P_L1_max) OR (0 <= #P_L2_max) OR (0 <= #P_L3_max) OR (0 <= #P_Total_max)) THEN
       #ZScale_End_P := #ZSCALE_END_SPQ1;
   ELSE
       ;
   END_IF;
   // selection maximum value
   #P := MAX(IN1 := #P_L1_max, IN2 := #P_L2_max, IN3 := #P_L3_max, IN4 := #P_Total_max, IN5 := 4.0);
   //
   #Scale_End_P := (REAL_TO_DINT(#P * #FACTOR)) + (#ZScale_End_P - (REAL_TO_DINT(#P * #FACTOR) MOD #ZScale_End_P));
   // calculate scale final reactive power max
   IF ((#AREA_TO_THOUSAND < #Q_L1_max) OR (#AREA_TO_THOUSAND < #Q_L2_max) OR
       (#AREA_TO_THOUSAND < #Q_L3_max) OR (#AREA_TO_THOUSAND < #Q_Total_max) OR
       (- #AREA_TO_THOUSAND > #Q_L1_min) OR (- #AREA_TO_THOUSAND > #Q_L2_min) OR
       (- #AREA_TO_THOUSAND > #Q_L3_min) OR (- #AREA_TO_THOUSAND > #Q_Total_min)) THEN
       #ZScale_End_Q := #ZSCALE_END_SPQ4;
   ELSIF ((#AREA_TO_HUNDRED < #Q_L1_max) OR (#AREA_TO_HUNDRED < #Q_L2_max) OR
       (#AREA_TO_HUNDRED < #Q_L3_max) OR (#AREA_TO_HUNDRED < #Q_Total_max) OR
       (- #AREA_TO_HUNDRED > #Q_L1_min) OR (- #AREA_TO_HUNDRED > #Q_L2_min) OR
       (- #AREA_TO_HUNDRED > #Q_L3_min) OR (- #AREA_TO_HUNDRED > #Q_Total_min)) THEN
       #ZScale_End_Q := #ZSCALE_END_SPQ3;
   ELSIF ((#AREA_TO_TEN < #Q_L1_max) OR (#AREA_TO_TEN < #Q_L2_max) OR
       (#AREA_TO_TEN < #Q_L3_max) OR (#AREA_TO_TEN < #Q_Total_max) OR
       (- #AREA_TO_TEN > #Q_L1_min) OR (- #AREA_TO_TEN > #Q_L2_min) OR
       (- #AREA_TO_TEN > #Q_L3_min) OR (- #AREA_TO_TEN > #Q_Total_min)) THEN
       #ZScale_End_Q := #ZSCALE_END_SPQ2;
   ELSIF ((0 <= #Q_L1_max) OR (0 <= #Q_L2_max) OR (0 <= #Q_L3_max) OR (0 <= #Q_Total_max) OR
       (0 >= #Q_L1_min) OR (0 >= #Q_L2_min) OR (0 >= #Q_L3_min) OR (0 >= #Q_Total_min)) THEN
       #ZScale_End_Q := #ZSCALE_END_SPQ1;
   ELSE
       ;
   END_IF;
   // calculate scale final reactive power max
   IF ((MAX(IN1 := #Q_L1_max, IN2 := #Q_L2_max, IN3 := #Q_L3_max, IN4 := #Q_Total_max)) = 0) THEN
       #Q := 4.0;
   ELSE
       #Q := MAX(IN1 := #Q_L1_max, IN2 := #Q_L2_max, IN3 := #Q_L3_max, IN4 := #Q_Total_max);
   END_IF;
   //
   IF (#Q > 0) THEN
       #Scale_End_Q := (REAL_TO_DINT(#Q * #FACTOR)) + (#ZScale_End_Q - (REAL_TO_DINT(#Q * #FACTOR) MOD #ZScale_End_Q));
   ELSIF (#Q < 0) THEN
       #Scale_End_Q := (REAL_TO_DINT(#Q * #FACTOR)) - (#ZScale_End_Q - (REAL_TO_DINT(#Q * #FACTOR) MOD #ZScale_End_Q));
   ELSE
       ;
   END_IF;
   // calculate scale final reactive power min
   IF ((MIN(IN1 := #Q_L1_min, IN2 := #Q_L2_min, IN3 := #Q_L3_min, IN4 := #Q_Total_min)) = 0) THEN
       #Q_min := -4.0;
   ELSE
       #Q_min := MIN(IN1 := #Q_L1_min, IN2 := #Q_L2_min, IN3 := #Q_L3_min, IN4 := #Q_Total_min);
   END_IF;
   //
   IF (#Q_min > 0) THEN
       #Scale_Begin_Q := 0;
   ELSIF (#Q_min < 0) THEN
       #Scale_Begin_Q := (REAL_TO_DINT(#Q_min * #FACTOR)) - (#ZScale_End_Q - (REAL_TO_DINT(#Q_min * #FACTOR) MOD #ZScale_End_Q));
   END_IF;
   //======================================================================================================================
   //==========value to output value=======================================================================================
   //======================================================================================================================
   // calculation value
   #Calculate_Value1 := #Driver_Data.Calculate_Value1;               // calculate value 1
   #Calculate_Value2 := #Driver_Data.Calculate_Value2;               // calculate value 2
   #Calculate_Value3 := #Driver_Data.Calculate_Value3;               // calculate value 3
   #Calculate_Value4 := #Driver_Data.Calculate_Value4;               // calculate value 4
   #Calculate_Value5 := #Driver_Data.Calculate_Value5;               // calculate value 5
   #Calculate_Value6 := #Driver_Data.Calculate_Value6;               // calculate value 6
   // selection of show modification
   #U_PH_PH_Mod := #Driver_Data.U_PH_PH_Mod;                    // voltage PH-PH show modification
   #U_PH_N_Mod := #Driver_Data.U_PH_N_Mod;                     // voltage PH-N show modification
   #I_Mod := #Driver_Data.I_Mod;                          // current show modification
   #S_Mod := #Driver_Data.S_Mod;                          // apparent power show modification
   #P_Mod := #Driver_Data.P_Mod;                          // active power show modification
   #Q_Mod := #Driver_Data.Q_Mod;                          // reactive power show modification
   #E_Mod := #Driver_Data.E_Mod;                          // energy meter show modification
   #f_Mod := #Driver_Data.f_Mod;                          // frequenz show modification
   #Cos_Mod := #Driver_Data.Cos_Mod;                        // efficiency factor show modification  
   // temp value to output value
   #f := #Zf;                                         // frequency
   #f_min := #Zf_min;                                     // minimum frequenz
   #f_max := #Zf_max;                                     // maximum frequenz
   #Cos_Total := #ZCos_Total;                                 // total efficiency factor
   #Cos_Total_min := #ZCos_Total_min;                             // minimum total efficiency factor
   #Cos_Total_max := #ZCos_Total_max;                             // maximum total efficiency factor
   #Cos_L1 := #ZCos_L1;                                    // efficiency factor L1       
   #Cos_L1_min := #ZCos_L1_min;                                // minimum efficiency factor L1
   #Cos_L1_max := #ZCos_L1_max;                                // maximum efficiency factor L1
   #Cos_L2 := #ZCos_L2;                                    // efficiency factor L2
   #Cos_L2_min := #ZCos_L2_min;                                // minimum efficiency factor L2
   #Cos_L2_max := #ZCos_L2_max;                                // maximum efficiency factor L2
   #Cos_L3 := #ZCOS_L3;                                    // efficiency factor L3
   #Cos_L3_min := #ZCos_L3_min;                                // minimum efficiency factor L3
   #Cos_L3_max := #ZCos_L3_max;                                // maximum efficiency factor L3
   // reset time Energy  
   #RTime_Data_Energy := #Driver_Data.RTime_Data_Energy;              // Reset Time
   #R_Year_Energy := BCD16_TO_INT(#ZRTime_Data_Energy[1]) + 100;      // Reset year   
   #R_Month_Energy := BCD16_TO_INT(#ZRTime_Data_Energy[2]) + 100;      // Reset month
   #R_Day_Energy := BCD16_TO_INT(#ZRTime_Data_Energy[3]) + 100;      // Reset day    
   #R_Hour_Energy := BCD16_TO_INT(#ZRTime_Data_Energy[4]) + 100;      // Reset hour   
   #R_Minute_Energy := BCD16_TO_INT(#ZRTime_Data_Energy[5]) + 100;      // Reset minute 
   #R_Second_Energy := BCD16_TO_INT(#ZRTime_Data_Energy[6]) + 100;      // Reset Second
   // reset time value
   #RTime_Data_Value := #Driver_Data.RTime_Data_Value;               // Reset Time
   #R_Year_Value := BCD16_TO_INT(#ZRTime_Data_Value[1]) + 100;       // Reset year   
   #R_Month_Value := BCD16_TO_INT(#ZRTime_Data_Value[2]) + 100;       // Reset month  
   #R_Day_Value := BCD16_TO_INT(#ZRTime_Data_Value[3]) + 100;       // Reset day    
   #R_Hour_Value := BCD16_TO_INT(#ZRTime_Data_Value[4]) + 100;       // Reset hour   
   #R_Minute_Value := BCD16_TO_INT(#ZRTime_Data_Value[5]) + 100;       // Reset minute 
   #R_Second_Value := BCD16_TO_INT(#ZRTime_Data_Value[6]) + 100;       // Reset Second
   // HMI_Bits
   IF (#Driver_Data.Rest_Start_Auto = TRUE) THEN
       #Start_Auto := FALSE;
       #Start_Acyclic := FALSE;
   ELSE
       ;
   END_IF;
   #HMI_Bits.Start_Acyclic := #Start_Acyclic;
   #HMI_Bits.Start_Auto := #Start_Auto;
   #HMI_Bits.Reset_min_max_Data := #Reset_min_max_Data;
   #HMI_Bits.Reset_Energy_Meter := #Reset_Energy_Meter;
   //
   #Read_Value := #Driver_Data.Read_Value;
   //======================================================================================================================
   //==========error code==================================================================================================
   //======================================================================================================================  
   // error code output
   #ERROR := #Fehler;
END_FUNCTION_BLOCK

FUNCTION_BLOCK "LAnInput6Lim"   // FB1750, FBD
TITLE = LAnInput6Lim
{ S7_Optimized_Access := 'FALSE' }
AUTHOR : VCC
FAMILY : ProcEqp
NAME : AnInput
VERSION : 1.0
// ================================================================================
// This module is used to read an analogue Input value and scale it. 
// It also gives the possibility to define 6 limits (High High High, High High, 
// High, Low, Low Low and Low Low Low level) and to create 6 alarms for these 
// limits. 
// ================================================================================
// stored: AutoNumber false, IsIECCheckEnabled false, SetENOAutomatically False, UDAEnableTagReadback false
   VAR_INPUT
      I_AnInput { ExternalAccessible := 'False'; ExternalVisible := 'False'; ExternalWritable := 'False'} : Real;   // Analogue Input Value
      I_MotorActive { ExternalAccessible := 'False'; ExternalVisible := 'False'; ExternalWritable := 'False'} : Bool;
      I_EnHHHAlarm { ExternalAccessible := 'False'; ExternalVisible := 'False'; ExternalWritable := 'False'} : Bool;   // Enable HHH Limit Alarm
      I_ResHHHAlarm { ExternalAccessible := 'False'; ExternalVisible := 'False'; ExternalWritable := 'False'} : Bool;   // Reset HHH Limit Alarm
      I_EnHHAlarm { ExternalAccessible := 'False'; ExternalVisible := 'False'; ExternalWritable := 'False'} : Bool;   // Enable HH Limit Alarm
      I_ResHHAlarm { ExternalAccessible := 'False'; ExternalVisible := 'False'; ExternalWritable := 'False'} : Bool;   // Reset HH Limit Alarm
      I_EnHAlarm { ExternalAccessible := 'False'; ExternalVisible := 'False'; ExternalWritable := 'False'} : Bool;   // Enable H Limit Alarm
      I_ResHAlarm { ExternalAccessible := 'False'; ExternalVisible := 'False'; ExternalWritable := 'False'} : Bool;   // Reset H Limit Alarm
      I_EnLAlarm { ExternalAccessible := 'False'; ExternalVisible := 'False'; ExternalWritable := 'False'} : Bool;   // Enable L Limit Alarm
      I_ResLAlarm { ExternalAccessible := 'False'; ExternalVisible := 'False'; ExternalWritable := 'False'} : Bool;   // Reset L Limit Alarm
      I_EnLLAlarm { ExternalAccessible := 'False'; ExternalVisible := 'False'; ExternalWritable := 'False'} : Bool;   // Enable LL Limit Alarm
      I_ResLLAlarm { ExternalAccessible := 'False'; ExternalVisible := 'False'; ExternalWritable := 'False'} : Bool;   // Reset LL Limit Alarm
      I_EnLLLAlarm { ExternalAccessible := 'False'; ExternalVisible := 'False'; ExternalWritable := 'False'} : Bool;   // Enable LLL Limit Alarm
      I_ResLLLAlarm { ExternalAccessible := 'False'; ExternalVisible := 'False'; ExternalWritable := 'False'} : Bool;   // Reset LLL Limit Alarm
      I_AlarmResetPB { ExternalAccessible := 'False'; ExternalVisible := 'False'; ExternalWritable := 'False'} : Bool;   // Alarm reset PB
   END_VAR
   VAR_OUTPUT
      O_HHHAlarm { ExternalAccessible := 'False'; ExternalVisible := 'False'; ExternalWritable := 'False'} : Bool;   // HHH Limit Alarm
      O_HHAlarm { ExternalAccessible := 'False'; ExternalVisible := 'False'; ExternalWritable := 'False'} : Bool;   // HH Limit Alarm
      O_HAlarm { ExternalAccessible := 'False'; ExternalVisible := 'False'; ExternalWritable := 'False'} : Bool;   // H Limit Alarm
      O_LAlarm { ExternalAccessible := 'False'; ExternalVisible := 'False'; ExternalWritable := 'False'} : Bool;   // L Limit Alarm
      O_LLAlarm { ExternalAccessible := 'False'; ExternalVisible := 'False'; ExternalWritable := 'False'} : Bool;   // LL Limit Alarm
      O_LLLAlarm { ExternalAccessible := 'False'; ExternalVisible := 'False'; ExternalWritable := 'False'} : Bool;   // LLL Limit Alarm
      O_AnInputScaled : Real;   // Analogue Input value after scaling
      O_AlarmABCondition { ExternalAccessible := 'False'; ExternalVisible := 'False'; ExternalWritable := 'False'} : Bool;   // Alarm AB condition
      O_HHHReached { ExternalAccessible := 'False'; ExternalVisible := 'False'; ExternalWritable := 'False'} : Bool;   // High High High Limit Reached
      O_HHReached { ExternalAccessible := 'False'; ExternalVisible := 'False'; ExternalWritable := 'False'} : Bool;   // High High Limit Reached
      O_HReached { ExternalAccessible := 'False'; ExternalVisible := 'False'; ExternalWritable := 'False'} : Bool;   // High Limit Reached
      O_LReached { ExternalAccessible := 'False'; ExternalVisible := 'False'; ExternalWritable := 'False'} : Bool;   // Low Limit Reached
      O_LLReached { ExternalAccessible := 'False'; ExternalVisible := 'False'; ExternalWritable := 'False'} : Bool;   // Low Low Limit Reached
      O_LLLReached { ExternalAccessible := 'False'; ExternalVisible := 'False'; ExternalWritable := 'False'} : Bool;   // Low Low Low Limit Reached
      H_IAnim { ExternalAccessible := 'False'; ExternalVisible := 'False'; ExternalWritable := 'False'} : DWord;   // HMI Animation of the icon
   END_VAR
   VAR DB_SPECIFIC
      H_In : Struct   // HMI
         AnInput_HighLimit : Real;   // From HMI : High Limit For Scaling Analogue Input
         AnInput_LowLimit : Real;   // From HMI : Low Limit For Scaling Analogue Input
         HHysteresis : Real;   // From HMI : Hysteresis value for High Limits
         LHysteresis : Real;   // From HMI : Hysteresis value for Low Limits
         HHHLimitValue : Real;   // From HMI : High High High Limit Value
         HHLimitValue : Real;   // From HMI : High High Limit Value
         HLimitValue : Real;   // From HMI : High Limit Value
         LLimitValue : Real;   // From HMI : Low Limit Value
         LLLimitValue : Real;   // From HMI : Low Low Limit Value
         LLLLimitValue : Real;   // From HMI : Low Low Low Limit Value
         TimeDelay : DInt;   // From HMI : Time delay for limits
         Forcing : Bool;   // From HMI : True if forced value must be used
         ForcedAnInput : Real;   // From HMI : Forced Analogue Input Value
      END_STRUCT;
      H_Out : Struct   // HMI
         Anim : Word;   // HMI Animation of the object
         DBnr : Int;   // HMI Animation DB number
      END_STRUCT;
   END_VAR
   VAR
      HHHLimitTimer { ExternalAccessible := 'False'; ExternalVisible := 'False'; ExternalWritable := 'False'; S7_SetPoint := 'True'} : "LTimer";   // Timer HHH Limit
      HHLimitTimer { ExternalAccessible := 'False'; ExternalVisible := 'False'; ExternalWritable := 'False'; S7_SetPoint := 'True'} : "LTimer";   // Timer HH Limit
      HLimitTimer { ExternalAccessible := 'False'; ExternalVisible := 'False'; ExternalWritable := 'False'; S7_SetPoint := 'True'} : "LTimer";   // Timer H Limit
      LLimitTimer { ExternalAccessible := 'False'; ExternalVisible := 'False'; ExternalWritable := 'False'; S7_SetPoint := 'True'} : "LTimer";   // Timer L Limit
      LLLimitTimer { ExternalAccessible := 'False'; ExternalVisible := 'False'; ExternalWritable := 'False'; S7_SetPoint := 'True'} : "LTimer";   // Timer LL Limit
      LLLLimitTimer { ExternalAccessible := 'False'; ExternalVisible := 'False'; ExternalWritable := 'False'; S7_SetPoint := 'True'} : "LTimer";   // Timer LLL Limit
   END_VAR
   VAR DB_SPECIFIC
      AnInputScaled { ExternalAccessible := 'False'; ExternalVisible := 'False'; ExternalWritable := 'False'} : Real;   // Analogue Input value after scaling
      HHHTempSR { ExternalAccessible := 'False'; ExternalVisible := 'False'; ExternalWritable := 'False'} : Bool;   // Temp variable for SET/RESET
      HHTempSR { ExternalAccessible := 'False'; ExternalVisible := 'False'; ExternalWritable := 'False'} : Bool;   // Temp variable for SET/RESET
      HTempSR { ExternalAccessible := 'False'; ExternalVisible := 'False'; ExternalWritable := 'False'} : Bool;   // Temp variable for SET/RESET
      LTempSR { ExternalAccessible := 'False'; ExternalVisible := 'False'; ExternalWritable := 'False'} : Bool;   // Temp variable for SET/RESET
      LLTempSR { ExternalAccessible := 'False'; ExternalVisible := 'False'; ExternalWritable := 'False'} : Bool;   // Temp variable for SET/RESET
      LLLTempSR { ExternalAccessible := 'False'; ExternalVisible := 'False'; ExternalWritable := 'False'} : Bool;   // Temp variable for SET/RESET
      HHHlimitHyst { ExternalAccessible := 'False'; ExternalVisible := 'False'; ExternalWritable := 'False'} : Real;   // HHH Limit with Hysteresis
      HHlimitHyst { ExternalAccessible := 'False'; ExternalVisible := 'False'; ExternalWritable := 'False'} : Real;   // HH Limit with Hysteresis
      HlimitHyst { ExternalAccessible := 'False'; ExternalVisible := 'False'; ExternalWritable := 'False'} : Real;   // H Limit with Hysteresis
      LlimitHyst { ExternalAccessible := 'False'; ExternalVisible := 'False'; ExternalWritable := 'False'} : Real;   // L Limit with Hysteresis
      LLlimitHyst { ExternalAccessible := 'False'; ExternalVisible := 'False'; ExternalWritable := 'False'} : Real;   // LL Limit with Hysteresis
      LLLlimitHyst { ExternalAccessible := 'False'; ExternalVisible := 'False'; ExternalWritable := 'False'} : Real;   // LLL Limit with Hysteresis
      HHHReached { ExternalAccessible := 'False'; ExternalVisible := 'False'; ExternalWritable := 'False'} : Bool;   // Temp variable HHH Limit Reached
      HHReached { ExternalAccessible := 'False'; ExternalVisible := 'False'; ExternalWritable := 'False'} : Bool;   // Temp variable HH Limit Reached
      HReached { ExternalAccessible := 'False'; ExternalVisible := 'False'; ExternalWritable := 'False'} : Bool;   // Temp variable H Limit Reached
      LReached { ExternalAccessible := 'False'; ExternalVisible := 'False'; ExternalWritable := 'False'} : Bool;   // Temp variable L Limit Reached
      LLReached { ExternalAccessible := 'False'; ExternalVisible := 'False'; ExternalWritable := 'False'} : Bool;   // Temp variable LL Limit Reached
      LLLReached { ExternalAccessible := 'False'; ExternalVisible := 'False'; ExternalWritable := 'False'} : Bool;   // Temp variable LLL Limit Reached
      HHHAlarmAlmCond { ExternalAccessible := 'False'; ExternalVisible := 'False'; ExternalWritable := 'False'} : Bool;   // HHHAlarm alarm condition
      HHAlarmAlmCond { ExternalAccessible := 'False'; ExternalVisible := 'False'; ExternalWritable := 'False'} : Bool;   // HHAlarm alarm condition
      HAlarmAlmCond { ExternalAccessible := 'False'; ExternalVisible := 'False'; ExternalWritable := 'False'} : Bool;   // HAlarm alarm condition
      LAlarmAlmCond { ExternalAccessible := 'False'; ExternalVisible := 'False'; ExternalWritable := 'False'} : Bool;   // LAlarm alarm condition
      LLAlarmAlmCond { ExternalAccessible := 'False'; ExternalVisible := 'False'; ExternalWritable := 'False'} : Bool;   // LLAlarm alarm condition
      LLLAlarmAlmCond { ExternalAccessible := 'False'; ExternalVisible := 'False'; ExternalWritable := 'False'} : Bool;   // LLLAlarm alarm condition
      HHHAlarm { ExternalAccessible := 'False'; ExternalVisible := 'False'; ExternalWritable := 'False'} : Bool;   // HHH Limit Alarm
      HHAlarm { ExternalAccessible := 'False'; ExternalVisible := 'False'; ExternalWritable := 'False'} : Bool;   // HH Limit Alarm
      HAlarm { ExternalAccessible := 'False'; ExternalVisible := 'False'; ExternalWritable := 'False'} : Bool;   // H Limit Alarm
      LAlarm { ExternalAccessible := 'False'; ExternalVisible := 'False'; ExternalWritable := 'False'} : Bool;   // L Limit Alarm
      LLAlarm { ExternalAccessible := 'False'; ExternalVisible := 'False'; ExternalWritable := 'False'} : Bool;   // LL Limit Alarm
      LLLAlarm { ExternalAccessible := 'False'; ExternalVisible := 'False'; ExternalWritable := 'False'} : Bool;   // LLL Limit Alarm
      AnInputTmp { ExternalAccessible := 'False'; ExternalVisible := 'False'; ExternalWritable := 'False'} : Real;   // Analog input temporary
      DBnr { ExternalAccessible := 'False'; ExternalVisible := 'False'; ExternalWritable := 'False'} : Int;   // HMI DB number
   END_VAR
   VAR
      HHH_Alarm { ExternalAccessible := 'False'; ExternalVisible := 'False'; ExternalWritable := 'False'; S7_SetPoint := 'True'} : "L1AlarmMultiIn";
      HH_Alarm { ExternalAccessible := 'False'; ExternalVisible := 'False'; ExternalWritable := 'False'; S7_SetPoint := 'True'} : "L1AlarmMultiIn";
      H_Alarm { ExternalAccessible := 'False'; ExternalVisible := 'False'; ExternalWritable := 'False'; S7_SetPoint := 'True'} : "L1AlarmMultiIn";
      L_Alarm { ExternalAccessible := 'False'; ExternalVisible := 'False'; ExternalWritable := 'False'; S7_SetPoint := 'True'} : "L1AlarmMultiIn";
      LL_Alarm { ExternalAccessible := 'False'; ExternalVisible := 'False'; ExternalWritable := 'False'; S7_SetPoint := 'True'} : "L1AlarmMultiIn";
      LLL_Alarm { ExternalAccessible := 'False'; ExternalVisible := 'False'; ExternalWritable := 'False'; S7_SetPoint := 'True'} : "L1AlarmMultiIn";
   END_VAR
BEGIN

NETWORK
TITLE = **** 1 - Inputs **** DB number
// DB number
      L     DINO;
      T     #DBnr;

REGION Network 2: **** 2.2 - Alarms - Alarm generation **** Alarm High High High Limit
   // Alarm High High High Limit
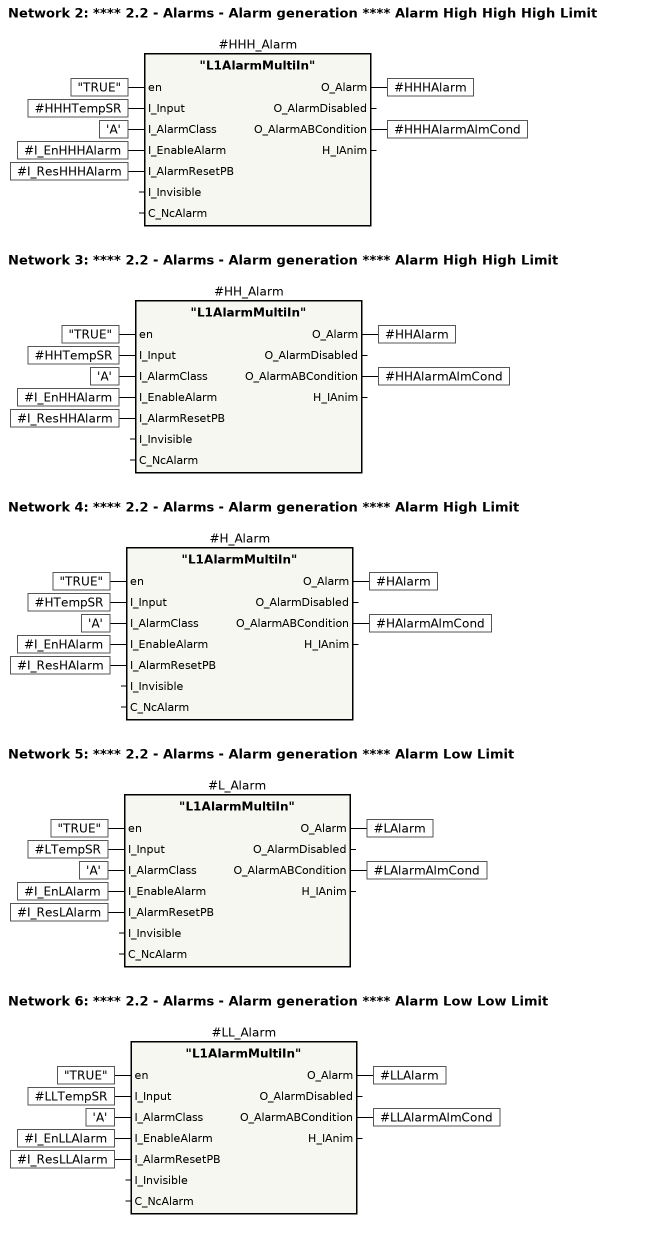
   IF "TRUE" THEN
       #HHH_Alarm(I_Input := #HHHTempSR,   // "L1AlarmMultiIn"
                  I_AlarmClass := 'A',
                  I_EnableAlarm := #I_EnHHHAlarm,
                  I_AlarmResetPB := #I_ResHHHAlarm,
                  O_Alarm => #HHHAlarm,
                  O_AlarmABCondition => #HHHAlarmAlmCond);
   END_IF;
END_REGION

REGION Network 3: **** 2.2 - Alarms - Alarm generation **** Alarm High High Limit
   // Alarm High High Limit
   IF "TRUE" THEN
       #HH_Alarm(I_Input := #HHTempSR,   // "L1AlarmMultiIn"
                 I_AlarmClass := 'A',
                 I_EnableAlarm := #I_EnHHAlarm,
                 I_AlarmResetPB := #I_ResHHAlarm,
                 O_Alarm => #HHAlarm,
                 O_AlarmABCondition => #HHAlarmAlmCond);
   END_IF;
END_REGION

REGION Network 4: **** 2.2 - Alarms - Alarm generation **** Alarm High Limit
   // Alarm High Limit
   IF "TRUE" THEN
       #H_Alarm(I_Input := #HTempSR,   // "L1AlarmMultiIn"
                I_AlarmClass := 'A',
                I_EnableAlarm := #I_EnHAlarm,
                I_AlarmResetPB := #I_ResHAlarm,
                O_Alarm => #HAlarm,
                O_AlarmABCondition => #HAlarmAlmCond);
   END_IF;
END_REGION

REGION Network 5: **** 2.2 - Alarms - Alarm generation **** Alarm Low Limit
   // Alarm Low Limit
   IF "TRUE" THEN
       #L_Alarm(I_Input := #LTempSR,   // "L1AlarmMultiIn"
                I_AlarmClass := 'A',
                I_EnableAlarm := #I_EnLAlarm,
                I_AlarmResetPB := #I_ResLAlarm,
                O_Alarm => #LAlarm,
                O_AlarmABCondition => #LAlarmAlmCond);
   END_IF;
END_REGION

REGION Network 6: **** 2.2 - Alarms - Alarm generation **** Alarm Low Low Limit
   // Alarm Low Low Limit
   IF "TRUE" THEN
       #LL_Alarm(I_Input := #LLTempSR,   // "L1AlarmMultiIn"
                 I_AlarmClass := 'A',
                 I_EnableAlarm := #I_EnLLAlarm,
                 I_AlarmResetPB := #I_ResLLAlarm,
                 O_Alarm => #LLAlarm,
                 O_AlarmABCondition => #LLAlarmAlmCond);
   END_IF;
END_REGION

REGION Network 7: **** 2.2 - Alarms - Alarm generation **** Alarm Low Low Low Limit
   // Alarm Low Low Low Limit
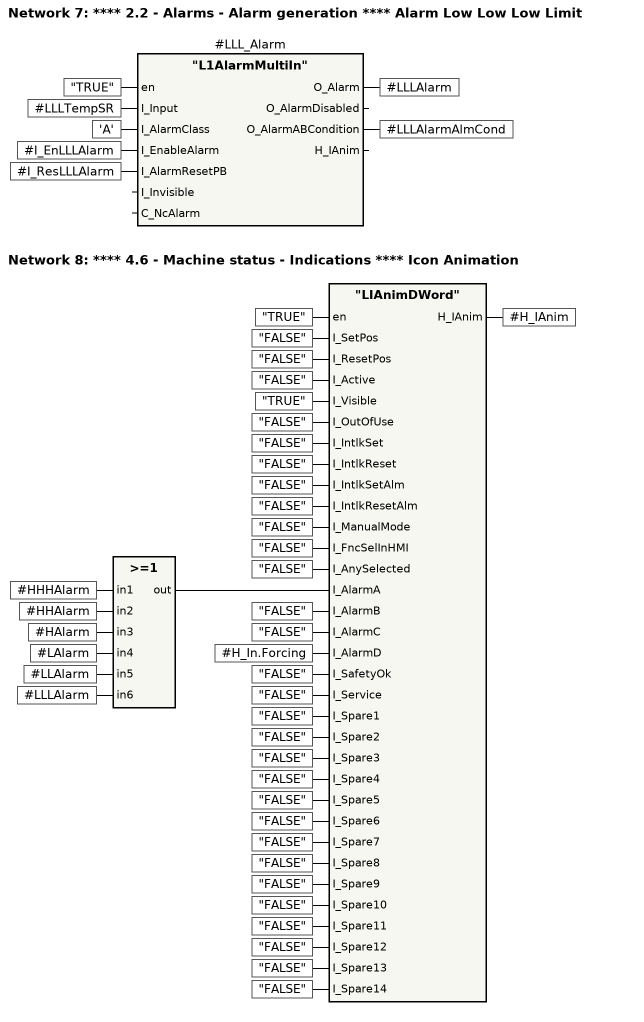
   IF "TRUE" THEN
       #LLL_Alarm(I_Input := #LLLTempSR,   // "L1AlarmMultiIn"
                  I_AlarmClass := 'A',
                  I_EnableAlarm := #I_EnLLLAlarm,
                  I_AlarmResetPB := #I_ResLLLAlarm,
                  O_Alarm => #LLLAlarm,
                  O_AlarmABCondition => #LLLAlarmAlmCond);
   END_IF;
END_REGION

REGION Network 8: **** 4.6 - Machine status - Indications **** Icon Animation
   // Icon Animation
   IF "TRUE" THEN
       "LIAnimDWord"(I_SetPos := "FALSE",
                     I_ResetPos := "FALSE",
                     I_Active := "FALSE",
                     I_Visible := "TRUE",
                     I_OutOfUse := "FALSE",
                     I_IntlkSet := "FALSE",
                     I_IntlkReset := "FALSE",
                     I_IntlkSetAlm := "FALSE",
                     I_IntlkResetAlm := "FALSE",
                     I_ManualMode := "FALSE",
                     I_FncSelInHMI := "FALSE",
                     I_AnySelected := "FALSE",
                     I_AlarmA := #HHHAlarm OR #HHAlarm OR #HAlarm OR #LAlarm OR #LLAlarm OR #LLLAlarm,
                     I_AlarmB := "FALSE",
                     I_AlarmC := "FALSE",
                     I_AlarmD := #H_In.Forcing,
                     I_SafetyOk := "FALSE",
                     I_Service := "FALSE",
                     I_Spare1 := "FALSE",
                     I_Spare2 := "FALSE",
                     I_Spare3 := "FALSE",
                     I_Spare4 := "FALSE",
                     I_Spare5 := "FALSE",
                     I_Spare6 := "FALSE",
                     I_Spare7 := "FALSE",
                     I_Spare8 := "FALSE",
                     I_Spare9 := "FALSE",
                     I_Spare10 := "FALSE",
                     I_Spare11 := "FALSE",
                     I_Spare12 := "FALSE",
                     I_Spare13 := "FALSE",
                     I_Spare14 := "FALSE",
                     H_IAnim => #H_IAnim);
   END_IF;
END_REGION

REGION Network 9: **** 4.6 - Machine status - Indications **** Animation
   // Animation
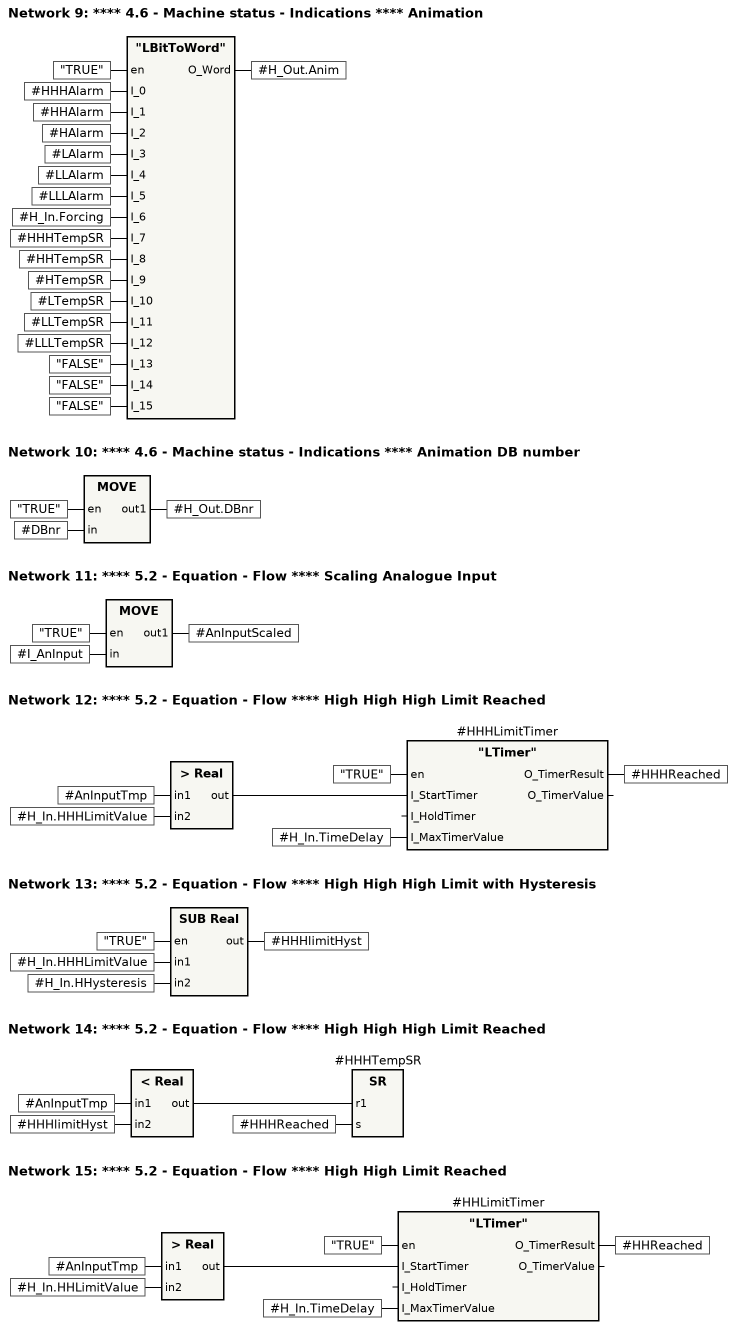
   IF "TRUE" THEN
       "LBitToWord"(I_0 := #HHHAlarm,
                    I_1 := #HHAlarm,
                    I_2 := #HAlarm,
                    I_3 := #LAlarm,
                    I_4 := #LLAlarm,
                    I_5 := #LLLAlarm,
                    I_6 := #H_In.Forcing,
                    I_7 := #HHHTempSR,
                    I_8 := #HHTempSR,
                    I_9 := #HTempSR,
                    I_10 := #LTempSR,
                    I_11 := #LLTempSR,
                    I_12 := #LLLTempSR,
                    I_13 := "FALSE",
                    I_14 := "FALSE",
                    I_15 := "FALSE",
                    O_Word => #H_Out.Anim);
   END_IF;
END_REGION

REGION Network 10: **** 4.6 - Machine status - Indications **** Animation DB number
   // Animation DB number
   IF "TRUE" THEN #H_Out.DBnr := #DBnr; END_IF;
END_REGION

REGION Network 11: **** 5.2 - Equation - Flow **** Scaling Analogue Input
   // Scaling Analogue Input
   IF "TRUE" THEN #AnInputScaled := #I_AnInput; END_IF;
END_REGION

REGION Network 12: **** 5.2 - Equation - Flow **** High High High Limit Reached
   // High High High Limit Reached
   IF "TRUE" THEN
       #HHHLimitTimer(I_StartTimer := #AnInputTmp > #H_In.HHHLimitValue,   // "LTimer"
                      I_MaxTimerValue := #H_In.TimeDelay,
                      O_TimerResult => #HHHReached);
   END_IF;
END_REGION

REGION Network 13: **** 5.2 - Equation - Flow **** High High High Limit with Hysteresis
   // High High High Limit with Hysteresis
   IF "TRUE" THEN #HHHlimitHyst := #H_In.HHHLimitValue - #H_In.HHysteresis; END_IF;
END_REGION

REGION Network 14: **** 5.2 - Equation - Flow **** High High High Limit Reached
   // High High High Limit Reached
   IF #HHHReached THEN
       #HHHTempSR := TRUE;   // SR flip-flop
   END_IF;
   IF #AnInputTmp < #HHHlimitHyst THEN #HHHTempSR := FALSE; END_IF;
END_REGION

REGION Network 15: **** 5.2 - Equation - Flow **** High High Limit Reached
   // High High Limit Reached
   IF "TRUE" THEN
       #HHLimitTimer(I_StartTimer := #AnInputTmp > #H_In.HHLimitValue,   // "LTimer"
                     I_MaxTimerValue := #H_In.TimeDelay,
                     O_TimerResult => #HHReached);
   END_IF;
END_REGION

REGION Network 16: **** 5.2 - Equation - Flow **** High High Limit with Hysteresis
   // High High Limit with Hysteresis
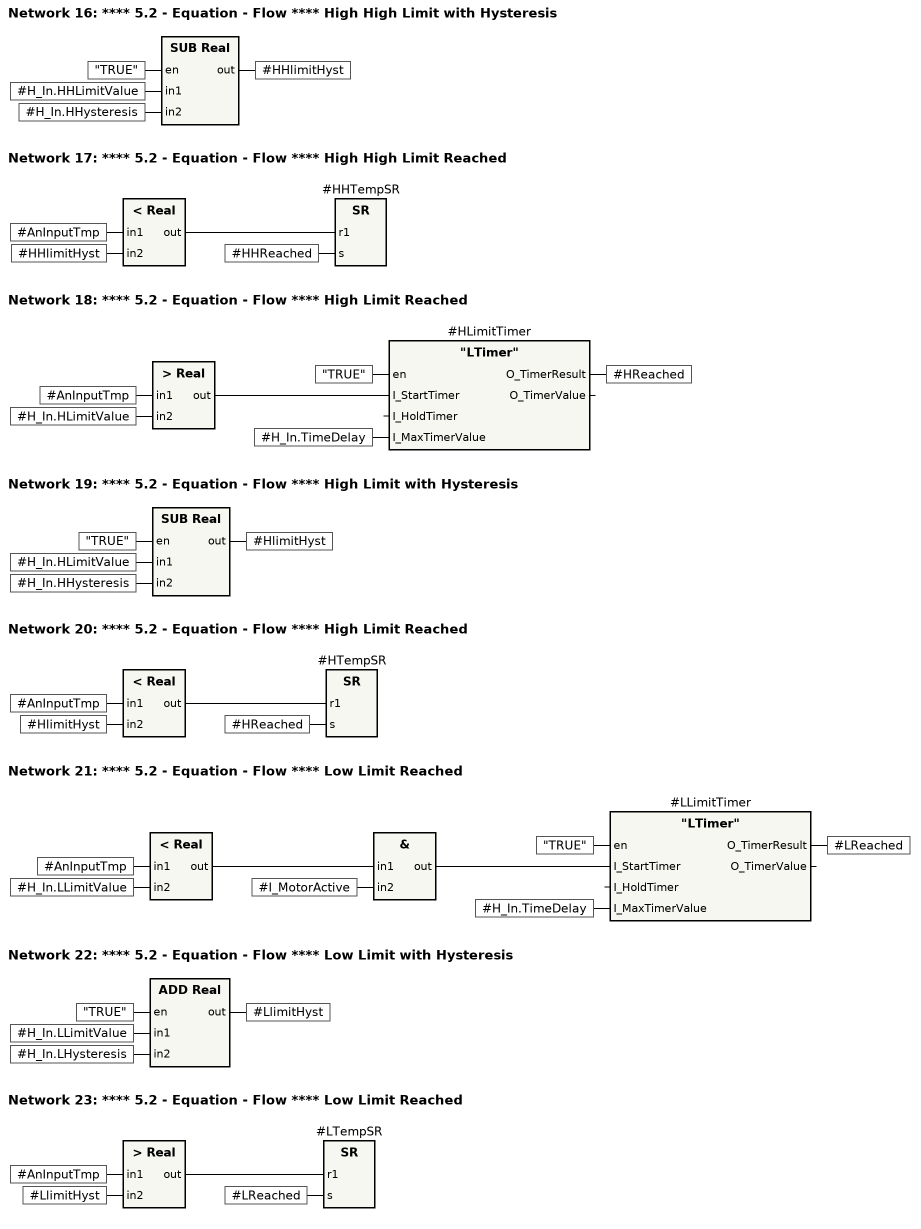
   IF "TRUE" THEN #HHlimitHyst := #H_In.HHLimitValue - #H_In.HHysteresis; END_IF;
END_REGION

REGION Network 17: **** 5.2 - Equation - Flow **** High High Limit Reached
   // High High Limit Reached
   IF #HHReached THEN
       #HHTempSR := TRUE;   // SR flip-flop
   END_IF;
   IF #AnInputTmp < #HHlimitHyst THEN #HHTempSR := FALSE; END_IF;
END_REGION

REGION Network 18: **** 5.2 - Equation - Flow **** High Limit Reached
   // High Limit Reached
   IF "TRUE" THEN
       #HLimitTimer(I_StartTimer := #AnInputTmp > #H_In.HLimitValue,   // "LTimer"
                    I_MaxTimerValue := #H_In.TimeDelay,
                    O_TimerResult => #HReached);
   END_IF;
END_REGION

REGION Network 19: **** 5.2 - Equation - Flow **** High Limit with Hysteresis
   // High Limit with Hysteresis
   IF "TRUE" THEN #HlimitHyst := #H_In.HLimitValue - #H_In.HHysteresis; END_IF;
END_REGION

REGION Network 20: **** 5.2 - Equation - Flow **** High Limit Reached
   // High Limit Reached
   IF #HReached THEN
       #HTempSR := TRUE;   // SR flip-flop
   END_IF;
   IF #AnInputTmp < #HlimitHyst THEN #HTempSR := FALSE; END_IF;
END_REGION

REGION Network 21: **** 5.2 - Equation - Flow **** Low Limit Reached
   // Low Limit Reached
   IF "TRUE" THEN
       #LLimitTimer(I_StartTimer := (#AnInputTmp < #H_In.LLimitValue) AND #I_MotorActive,   // "LTimer"
                    I_MaxTimerValue := #H_In.TimeDelay,
                    O_TimerResult => #LReached);
   END_IF;
END_REGION

REGION Network 22: **** 5.2 - Equation - Flow **** Low Limit with Hysteresis
   // Low Limit with Hysteresis
   IF "TRUE" THEN #LlimitHyst := #H_In.LLimitValue + #H_In.LHysteresis; END_IF;
END_REGION

REGION Network 23: **** 5.2 - Equation - Flow **** Low Limit Reached
   // Low Limit Reached
   IF #LReached THEN
       #LTempSR := TRUE;   // SR flip-flop
   END_IF;
   IF #AnInputTmp > #LlimitHyst THEN #LTempSR := FALSE; END_IF;
END_REGION

REGION Network 24: **** 5.2 - Equation - Flow **** Low Low Limit Reached
   // Low Low Limit Reached
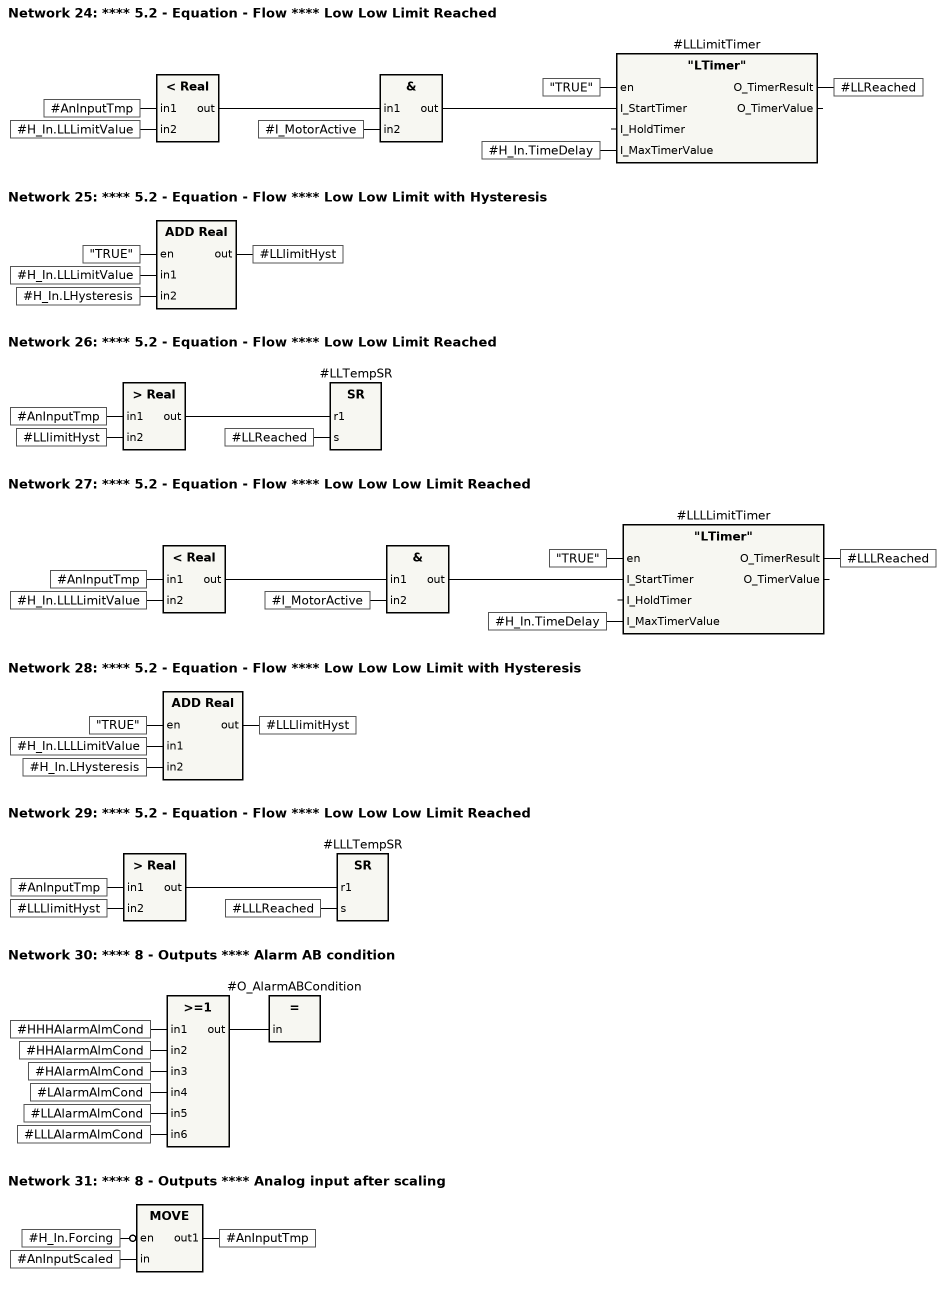
   IF "TRUE" THEN
       #LLLimitTimer(I_StartTimer := (#AnInputTmp < #H_In.LLLimitValue) AND #I_MotorActive,   // "LTimer"
                     I_MaxTimerValue := #H_In.TimeDelay,
                     O_TimerResult => #LLReached);
   END_IF;
END_REGION

REGION Network 25: **** 5.2 - Equation - Flow **** Low Low Limit with Hysteresis
   // Low Low Limit with Hysteresis
   IF "TRUE" THEN #LLlimitHyst := #H_In.LLLimitValue + #H_In.LHysteresis; END_IF;
END_REGION

REGION Network 26: **** 5.2 - Equation - Flow **** Low Low Limit Reached
   // Low Low Limit Reached
   IF #LLReached THEN
       #LLTempSR := TRUE;   // SR flip-flop
   END_IF;
   IF #AnInputTmp > #LLlimitHyst THEN #LLTempSR := FALSE; END_IF;
END_REGION

REGION Network 27: **** 5.2 - Equation - Flow **** Low Low Low Limit Reached
   // Low Low Low Limit Reached
   IF "TRUE" THEN
       #LLLLimitTimer(I_StartTimer := (#AnInputTmp < #H_In.LLLLimitValue) AND #I_MotorActive,   // "LTimer"
                      I_MaxTimerValue := #H_In.TimeDelay,
                      O_TimerResult => #LLLReached);
   END_IF;
END_REGION

REGION Network 28: **** 5.2 - Equation - Flow **** Low Low Low Limit with Hysteresis
   // Low Low Low Limit with Hysteresis
   IF "TRUE" THEN #LLLlimitHyst := #H_In.LLLLimitValue + #H_In.LHysteresis; END_IF;
END_REGION

REGION Network 29: **** 5.2 - Equation - Flow **** Low Low Low Limit Reached
   // Low Low Low Limit Reached
   IF #LLLReached THEN
       #LLLTempSR := TRUE;   // SR flip-flop
   END_IF;
   IF #AnInputTmp > #LLLlimitHyst THEN #LLLTempSR := FALSE; END_IF;
END_REGION

REGION Network 30: **** 8 - Outputs **** Alarm AB condition
   // Alarm AB condition
   #O_AlarmABCondition := #HHHAlarmAlmCond OR #HHAlarmAlmCond OR #HAlarmAlmCond OR #LAlarmAlmCond OR #LLAlarmAlmCond OR #LLLAlarmAlmCond;
END_REGION

REGION Network 31: **** 8 - Outputs **** Analog input after scaling
   // Analog input after scaling
   IF NOT #H_In.Forcing THEN #AnInputTmp := #AnInputScaled; END_IF;
END_REGION

REGION Network 32: **** 8 - Outputs **** Forcing Analogue Input
   // Forcing Analogue Input
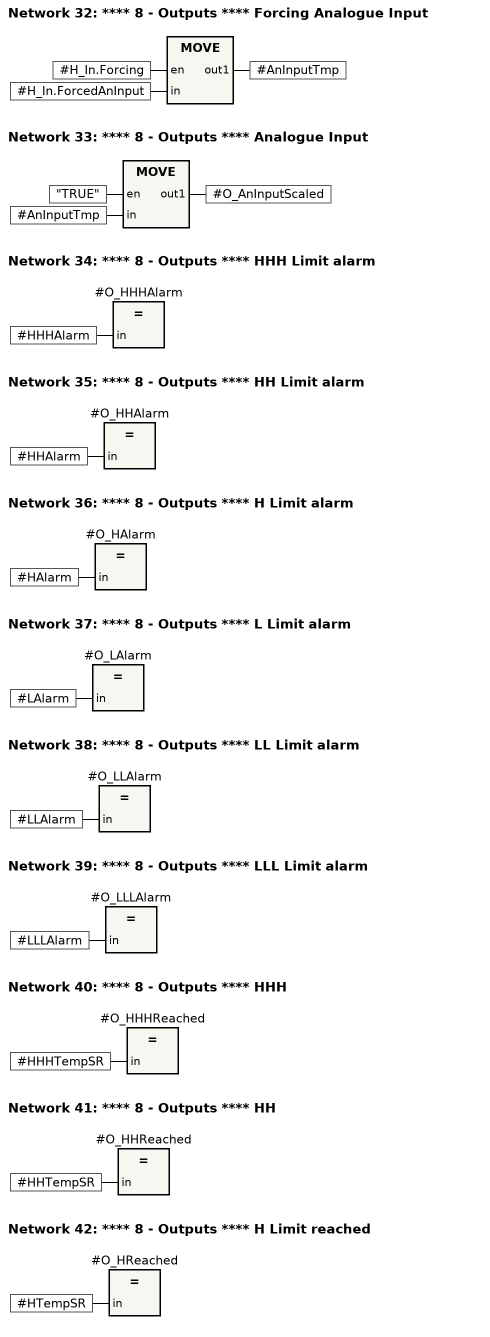
   IF #H_In.Forcing THEN #AnInputTmp := #H_In.ForcedAnInput; END_IF;
END_REGION

REGION Network 33: **** 8 - Outputs **** Analogue Input
   // Analogue Input
   IF "TRUE" THEN #O_AnInputScaled := #AnInputTmp; END_IF;
END_REGION

REGION Network 34: **** 8 - Outputs **** HHH Limit alarm
   // HHH Limit alarm
   #O_HHHAlarm := #HHHAlarm;
END_REGION

REGION Network 35: **** 8 - Outputs **** HH Limit alarm
   // HH Limit alarm
   #O_HHAlarm := #HHAlarm;
END_REGION

REGION Network 36: **** 8 - Outputs **** H Limit alarm
   // H Limit alarm
   #O_HAlarm := #HAlarm;
END_REGION

REGION Network 37: **** 8 - Outputs **** L Limit alarm
   // L Limit alarm
   #O_LAlarm := #LAlarm;
END_REGION

REGION Network 38: **** 8 - Outputs **** LL Limit alarm
   // LL Limit alarm
   #O_LLAlarm := #LLAlarm;
END_REGION

REGION Network 39: **** 8 - Outputs **** LLL Limit alarm
   // LLL Limit alarm
   #O_LLLAlarm := #LLLAlarm;
END_REGION

REGION Network 40: **** 8 - Outputs **** HHH
   // HHH
   //  Limit reached
   #O_HHHReached := #HHHTempSR;
END_REGION

REGION Network 41: **** 8 - Outputs **** HH
   // HH
   //  Limit reached
   #O_HHReached := #HHTempSR;
END_REGION

REGION Network 42: **** 8 - Outputs **** H Limit reached
   // H Limit reached
   #O_HReached := #HTempSR;
END_REGION

REGION Network 43: **** 8 - Outputs **** L Limit reached
   // L Limit reached
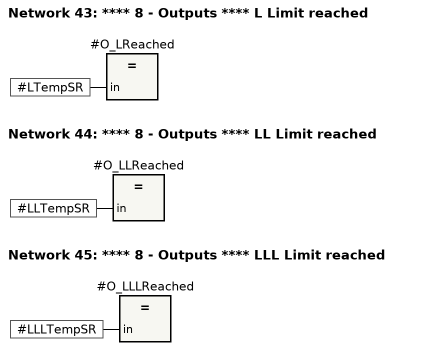
   #O_LReached := #LTempSR;
END_REGION

REGION Network 44: **** 8 - Outputs **** LL Limit reached
   // LL Limit reached
   #O_LLReached := #LLTempSR;
END_REGION

REGION Network 45: **** 8 - Outputs **** LLL Limit reached
   // LLL Limit reached
   #O_LLLReached := #LLLTempSR;
END_REGION
END_FUNCTION_BLOCK

FUNCTION_BLOCK "LCounter1Week"   // FB1801, FBD
TITLE = LCounter1Week
{ S7_Optimized_Access := 'FALSE' }
AUTHOR : VCC
FAMILY : Supervis
NAME : LCpt1W
VERSION : 1.0
// ==============================================================================
// Module create to count body produced during all shifts of the week.
// One counter per shift (moring - evening & night) per day (from monday to sunday)
// all total are foreseen.
// 
// --------------------------------------------------------------------
// Day          ! Morning shift ! Evening shift ! Night shift ! total !
// -------------!---------------!---------------!-------------!-------!
// Monday (1)   !               !               !             !       !
// -------------!---------------!---------------!-------------!-------!
// Tuesday (2)  !               !               !             !       !
// -------------!---------------!---------------!-------------!-------!
// Wednesday (3)!               !               !             !       !
// -------------!---------------!---------------!-------------!-------!
// Thursday (4) !               !               !             !       !
// -------------!---------------!---------------!-------------!-------!
// Friday (5)   !               !               !             !       !
// -------------!---------------!---------------!-------------!-------!
// Saturday (6) !               !               !             !       !
// -------------!---------------!---------------!-------------!-------!
// Sunday (7)   !               !               !             !       !
// ====================================================================
// Amount       !               !               !             !       !
// ====================================================================
// Tatal        !=============================================!       !
// ====================================================================
// 
// ==============================================================================
// stored: AutoNumber false, IsIECCheckEnabled false, SetENOAutomatically False, UDAEnableTagReadback false
   VAR_INPUT
      I_CountedInput { ExternalAccessible := 'False'; ExternalVisible := 'False'; ExternalWritable := 'False'} : Bool;   // Value to be counted
      I_MorningShift { ExternalAccessible := 'False'; ExternalVisible := 'False'; ExternalWritable := 'False'} : Bool;   // Morning shift
      I_EveningShift { ExternalAccessible := 'False'; ExternalVisible := 'False'; ExternalWritable := 'False'} : Bool;   // Evening shift
      I_NightShift { ExternalAccessible := 'False'; ExternalVisible := 'False'; ExternalWritable := 'False'} : Bool;   // NightShift
   END_VAR
   VAR_OUTPUT
      H_IAnim { ExternalAccessible := 'False'; ExternalVisible := 'False'; ExternalWritable := 'False'} : Word;   // HMI Animation of the icon
   END_VAR
   VAR DB_SPECIFIC
      H_Out : Struct   // HMI
         Anim : Word;   // HMI Animation of the object
         MorningDay1Value : Int;   // Total Production value Monday (day 1) - Morning Shift
         EveningDay1Value : Int;   // Total Production value Monday (day 1) - Evening Shift
         NightDay1Value : Int;   // Total Production value Monday (day 1) - Night Shift
         MorningDay2Value : Int;   // Total Production value Tuesday (day 2) - Morning Shift
         EveningDay2Value : Int;   // Total Production value Tuesday (day 2) - Evening Shift
         NightDay2Value : Int;   // Total Production value Tuesday (day 2) - Night Shift
         MorningDay3Value : Int;   // Total Production value Wednesday (day 3) - Morning Shift
         EveningDay3Value : Int;   // Total Production value Wednesday (day 3) - Evening Shift
         NightDay3Value : Int;   // Total Production value Wednesday (day 3) - Night Shift
         MorningDay4Value : Int;   // Total Production value Thursday (day 4) - Morning Shift
         EveningDay4Value : Int;   // Total Production value Thursday (day 4) - Evening Shift
         NightDay4Value : Int;   // Total Production value Thursday (day 4) - Night Shift
         MorningDay5Value : Int;   // Total Production value Friday (day 5) - Morning Shift
         EveningDay5Value : Int;   // Total Production value Friday (day 5) - Evening Shift
         NightDay5Value : Int;   // Total Production value Friday (day 5) - Night Shift
         MorningDay6Value : Int;   // Total Production value Saturday (day 6) - Morning Shift
         EveningDay6Value : Int;   // Total Production value Saturday (day 6) - Evening Shift
         NightDay6Value : Int;   // Total Production value Saturday (day 6) - Night Shift
         MorningDay7Value : Int;   // Production value Sunday (day 7) - Morning Shift
         EveningDay7Value : Int;   // Production value Sunday (day 7) - Evening Shift
         NightDay7Value : Int;   // Production value Sunday (day 7) - Night Shift
         Day1Value : Int;   // Total Production value Monday (day 1)
         Day2Value : Int;   // Total Production value tuesday (day 2)
         Day3Value : Int;   // Total Production value Wednesday (day 3)
         Day4Value : Int;   // Total Production value Thursday (day 4)
         Day5Value : Int;   // Total Production value Friday (day 5)
         Day6Value : Int;   // Total Production value Saturday (day 6)
         Day7Value : Int;   // Total Production value Sunday (day 7)
         TotalMorning : Int;   // Total Production value Morning
         TotalEvening : Int;   // Total Production value Evening
         TotalNight : Int;   // Total Production value Night
         WeekValue : Int;   // Total Production value Week
         TotalValue : DInt;   // Total production value
         DBnr : Int;   // HMI Animation DB number
      END_STRUCT;
      CountedInputPulse { ExternalAccessible := 'False'; ExternalVisible := 'False'; ExternalWritable := 'False'} : Bool;   // Pulse of value to be counted
      CountUp { ExternalAccessible := 'False'; ExternalVisible := 'False'; ExternalWritable := 'False'} : Bool;   // Pulse of value to be counted
      MorningShiftPulse { ExternalAccessible := 'False'; ExternalVisible := 'False'; ExternalWritable := 'False'} : Bool;   // Pulse of Morning shift
      MorningPulse { ExternalAccessible := 'False'; ExternalVisible := 'False'; ExternalWritable := 'False'} : Bool;   // Pulse of Morning shift
      Day1 { ExternalAccessible := 'False'; ExternalVisible := 'False'; ExternalWritable := 'False'} : Bool;   // Day 1 = Monday
      Day2 { ExternalAccessible := 'False'; ExternalVisible := 'False'; ExternalWritable := 'False'} : Bool;   // Day 2 = Tuesday
      Day3 { ExternalAccessible := 'False'; ExternalVisible := 'False'; ExternalWritable := 'False'} : Bool;   // Day 3 = Wednesday
      Day4 { ExternalAccessible := 'False'; ExternalVisible := 'False'; ExternalWritable := 'False'} : Bool;   // Day 4 = Thursday
      Day5 { ExternalAccessible := 'False'; ExternalVisible := 'False'; ExternalWritable := 'False'} : Bool;   // Day 5 = Friday
      Day6 { ExternalAccessible := 'False'; ExternalVisible := 'False'; ExternalWritable := 'False'} : Bool;   // Day 6 = Saturday
      Day7 { ExternalAccessible := 'False'; ExternalVisible := 'False'; ExternalWritable := 'False'} : Bool;   // Day 7 = Sunday
      MorningValue { ExternalAccessible := 'False'; ExternalVisible := 'False'; ExternalWritable := 'False'} : Int;   // Morning production value
      EveningValue { ExternalAccessible := 'False'; ExternalVisible := 'False'; ExternalWritable := 'False'} : Int;   // Evening production value
      NightValue { ExternalAccessible := 'False'; ExternalVisible := 'False'; ExternalWritable := 'False'} : Int;   // Night production value
      MorningDay1Value { ExternalAccessible := 'False'; ExternalVisible := 'False'; ExternalWritable := 'False'} : Int;   // Total Production value Monday (day 1) - Morning Shift
      EveningDay1Value { ExternalAccessible := 'False'; ExternalVisible := 'False'; ExternalWritable := 'False'} : Int;   // Total Production value Monday (day 1) - Evening Shift
      NightDay1Value { ExternalAccessible := 'False'; ExternalVisible := 'False'; ExternalWritable := 'False'} : Int;   // Total Production value Monday (day 1) - Night Shift
      MorningDay2Value { ExternalAccessible := 'False'; ExternalVisible := 'False'; ExternalWritable := 'False'} : Int;   // Total Production value Tuesday (day 2) - Morning Shift
      EveningDay2Value { ExternalAccessible := 'False'; ExternalVisible := 'False'; ExternalWritable := 'False'} : Int;   // Total Production value Tuesday (day 2) - Evening Shift
      NightDay2Value { ExternalAccessible := 'False'; ExternalVisible := 'False'; ExternalWritable := 'False'} : Int;   // Total Production value Tuesday (day 2) - Night Shift
      MorningDay3Value { ExternalAccessible := 'False'; ExternalVisible := 'False'; ExternalWritable := 'False'} : Int;   // Total Production value Wednesday (day 3) - Morning Shift
      EveningDay3Value { ExternalAccessible := 'False'; ExternalVisible := 'False'; ExternalWritable := 'False'} : Int;   // Total Production value Wednesday (day 3) - Evening Shift
      NightDay3Value { ExternalAccessible := 'False'; ExternalVisible := 'False'; ExternalWritable := 'False'} : Int;   // Total Production value Wednesday (day 3) - Night Shift
      MorningDay4Value { ExternalAccessible := 'False'; ExternalVisible := 'False'; ExternalWritable := 'False'} : Int;   // Total Production value Thursday (day 4) - Morning Shift
      EveningDay4Value { ExternalAccessible := 'False'; ExternalVisible := 'False'; ExternalWritable := 'False'} : Int;   // Total Production value Thursday (day 4) - Evening Shift
      NightDay4Value { ExternalAccessible := 'False'; ExternalVisible := 'False'; ExternalWritable := 'False'} : Int;   // Total Production value Thursday (day 4) - Night Shift
      MorningDay5Value { ExternalAccessible := 'False'; ExternalVisible := 'False'; ExternalWritable := 'False'} : Int;   // Total Production value Friday (day 5) - Morning Shift
      EveningDay5Value { ExternalAccessible := 'False'; ExternalVisible := 'False'; ExternalWritable := 'False'} : Int;   // Total Production value Friday (day 5) - Evening Shift
      NightDay5Value { ExternalAccessible := 'False'; ExternalVisible := 'False'; ExternalWritable := 'False'} : Int;   // Total Production value Friday (day 5) - Night Shift
      MorningDay6Value { ExternalAccessible := 'False'; ExternalVisible := 'False'; ExternalWritable := 'False'} : Int;   // Total Production value Saturday (day 6) - Morning Shift
      EveningDay6Value { ExternalAccessible := 'False'; ExternalVisible := 'False'; ExternalWritable := 'False'} : Int;   // Total Production value Saturday (day 6) - Evening Shift
      NightDay6Value { ExternalAccessible := 'False'; ExternalVisible := 'False'; ExternalWritable := 'False'} : Int;   // Total Production value Saturday (day 6) - Night Shift
      MorningDay7Value { ExternalAccessible := 'False'; ExternalVisible := 'False'; ExternalWritable := 'False'} : Int;   // Production value Sunday (day 7) - Morning Shift
      EveningDay7Value { ExternalAccessible := 'False'; ExternalVisible := 'False'; ExternalWritable := 'False'} : Int;   // Production value Sunday (day 7) - Evening Shift
      NightDay7Value { ExternalAccessible := 'False'; ExternalVisible := 'False'; ExternalWritable := 'False'} : Int;   // Production value Sunday (day 7) - Night Shift
      Day1Value { ExternalAccessible := 'False'; ExternalVisible := 'False'; ExternalWritable := 'False'} : Int;   // Total Production value Monday (day 1)
      Day2Value { ExternalAccessible := 'False'; ExternalVisible := 'False'; ExternalWritable := 'False'} : Int;   // Total Production value tuesday (day 2)
      Day3Value { ExternalAccessible := 'False'; ExternalVisible := 'False'; ExternalWritable := 'False'} : Int;   // Total Production value Wednesday (day 3)
      Day4Value { ExternalAccessible := 'False'; ExternalVisible := 'False'; ExternalWritable := 'False'} : Int;   // Total Production value Thursday (day 4)
      Day5Value { ExternalAccessible := 'False'; ExternalVisible := 'False'; ExternalWritable := 'False'} : Int;   // Total Production value Friday (day 5)
      Day6Value { ExternalAccessible := 'False'; ExternalVisible := 'False'; ExternalWritable := 'False'} : Int;   // Total Production value Saturday (day 6)
      Day7Value { ExternalAccessible := 'False'; ExternalVisible := 'False'; ExternalWritable := 'False'} : Int;   // Total Production value Sunday (day 7)
      WeekValue { ExternalAccessible := 'False'; ExternalVisible := 'False'; ExternalWritable := 'False'} : Int;   // Total Production value Week
      TotalValue { ExternalAccessible := 'False'; ExternalVisible := 'False'; ExternalWritable := 'False'} : DInt;   // Total production value
      DBnr { ExternalAccessible := 'False'; ExternalVisible := 'False'; ExternalWritable := 'False'} : Int;   // HMI DB number
   END_VAR
   VAR_TEMP   // added for the SCL form of the ladder/FBD networks
      _w1 : Bool;
   END_VAR
BEGIN

NETWORK
TITLE = **** 1 - Inputs **** DB number
// DB number
      L     DINO;
      T     #DBnr;

REGION Network 2: **** 4.4 - Machine status - Calculated **** Total production counter
   // Total production counter
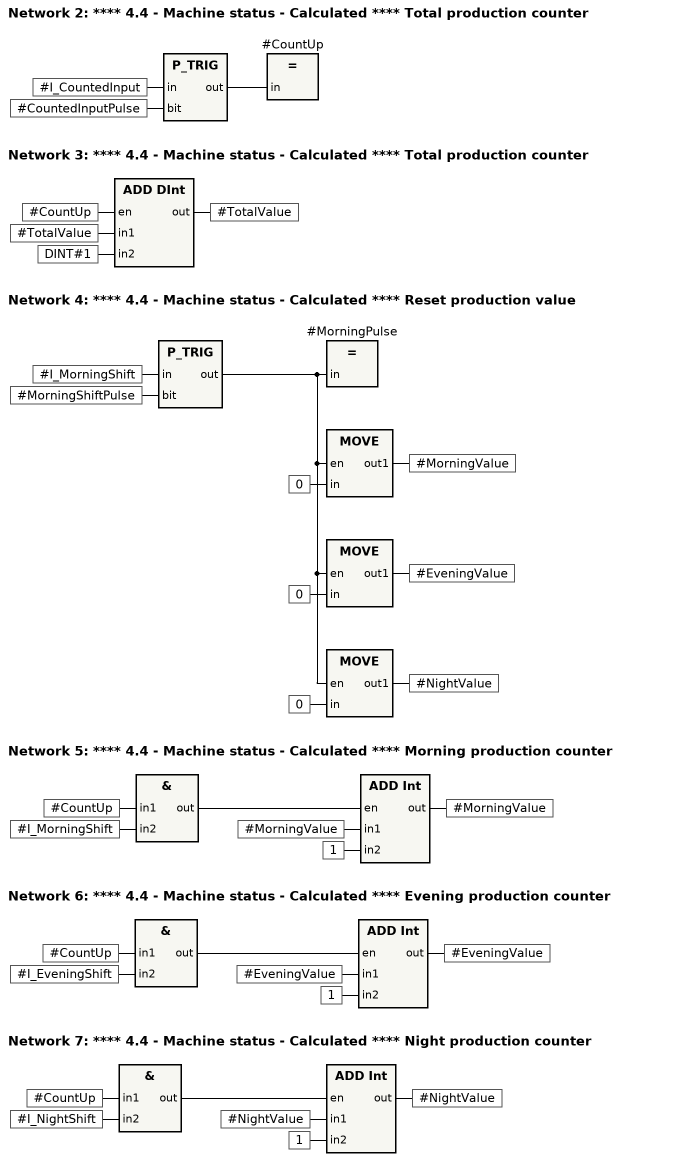
   #_w1 := #I_CountedInput AND NOT #CountedInputPulse;   // rising edge
   #CountedInputPulse := #I_CountedInput;
   #CountUp := #_w1;
END_REGION

REGION Network 3: **** 4.4 - Machine status - Calculated **** Total production counter
   // Total production counter
   IF #CountUp THEN #TotalValue := #TotalValue + DINT#1; END_IF;
END_REGION

REGION Network 4: **** 4.4 - Machine status - Calculated **** Reset production value
   // Reset production value
   #_w1 := #I_MorningShift AND NOT #MorningShiftPulse;   // rising edge
   #MorningShiftPulse := #I_MorningShift;
   #MorningPulse := #_w1;
   IF #_w1 THEN
       #MorningValue := 0;
       #EveningValue := 0;
       #NightValue := 0;
   END_IF;
END_REGION

REGION Network 5: **** 4.4 - Machine status - Calculated **** Morning production counter
   // Morning production counter
   IF #CountUp AND #I_MorningShift THEN #MorningValue := #MorningValue + 1; END_IF;
END_REGION

REGION Network 6: **** 4.4 - Machine status - Calculated **** Evening production counter
   // Evening production counter
   IF #CountUp AND #I_EveningShift THEN #EveningValue := #EveningValue + 1; END_IF;
END_REGION

REGION Network 7: **** 4.4 - Machine status - Calculated **** Night production counter
   // Night production counter
   IF #CountUp AND #I_NightShift THEN #NightValue := #NightValue + 1; END_IF;
END_REGION

REGION Network 8: **** 4.4 - Machine status - Calculated **** Set Monday - reset other days
   // Set Monday - reset other days
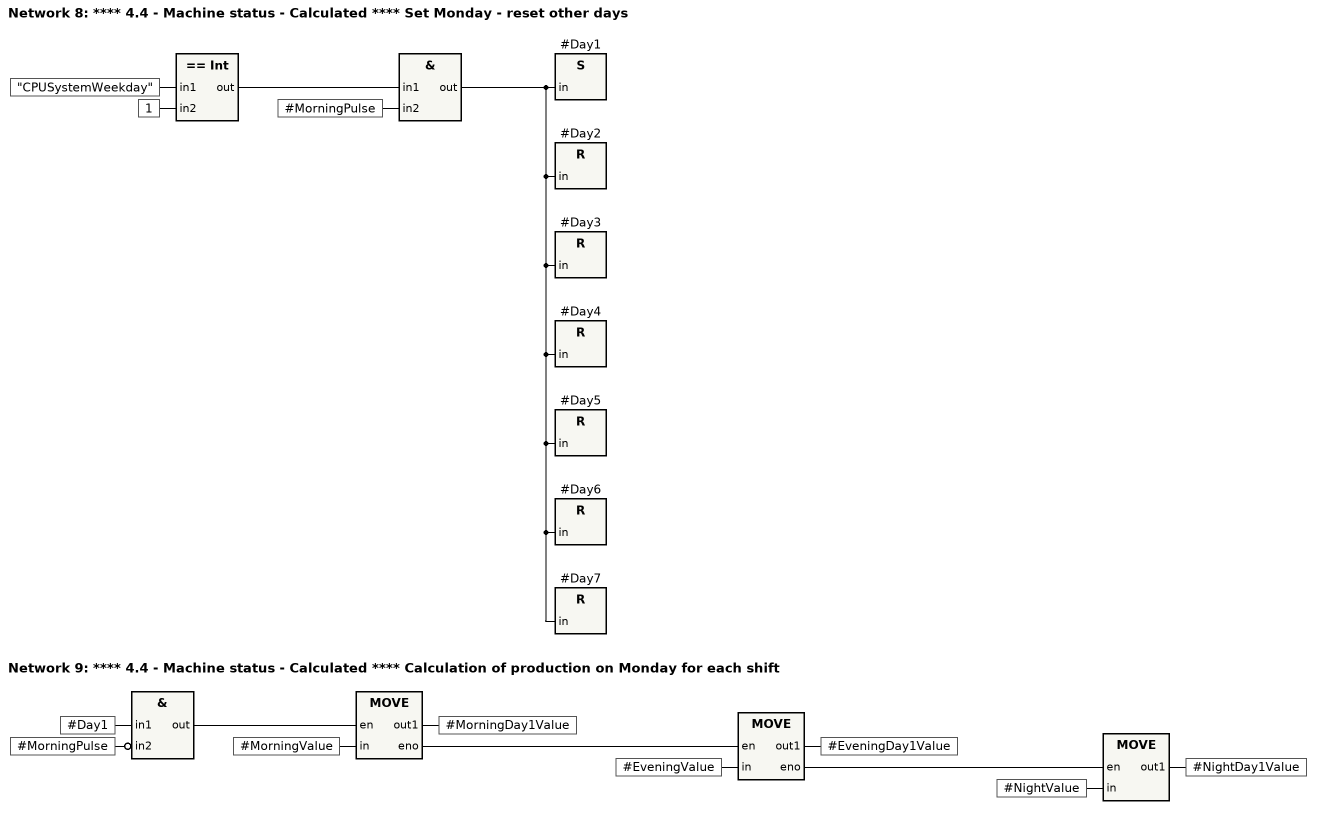
   IF ("CPUSystemWeekday" = 1) AND #MorningPulse THEN
       #Day1 := TRUE;
       #Day2 := FALSE;
       #Day3 := FALSE;
       #Day4 := FALSE;
       #Day5 := FALSE;
       #Day6 := FALSE;
       #Day7 := FALSE;
   END_IF;
END_REGION

REGION Network 9: **** 4.4 - Machine status - Calculated **** Calculation of production on Monday for each shift
   // Calculation of production on Monday for each shift
   // ENO of a box is taken as its EN; it also drops when the box reports an error
   IF #Day1 AND NOT #MorningPulse THEN
       #MorningDay1Value := #MorningValue;
       #EveningDay1Value := #EveningValue;
       #NightDay1Value := #NightValue;
   END_IF;
END_REGION

NETWORK
TITLE = **** 4.4 - Machine status - Calculated **** Total production on Monday
// Total production on Monday
      L     #MorningDay1Value;  // amount of bodies on day 1 - Morning shift (Monday)
      L     #EveningDay1Value;  // amount of bodies on day 1 - Evening shift (Monday)
      +I;
      L     #NightDay1Value;  // amount of bodies on day 1 - Night shift (Monday)
      +I;
      T     #Day1Value;  // amount of bodies on day 1 (Monday)

REGION Network 11: **** 4.4 - Machine status - Calculated **** Set Tuesday - reset other days
   // Set Tuesday - reset other days
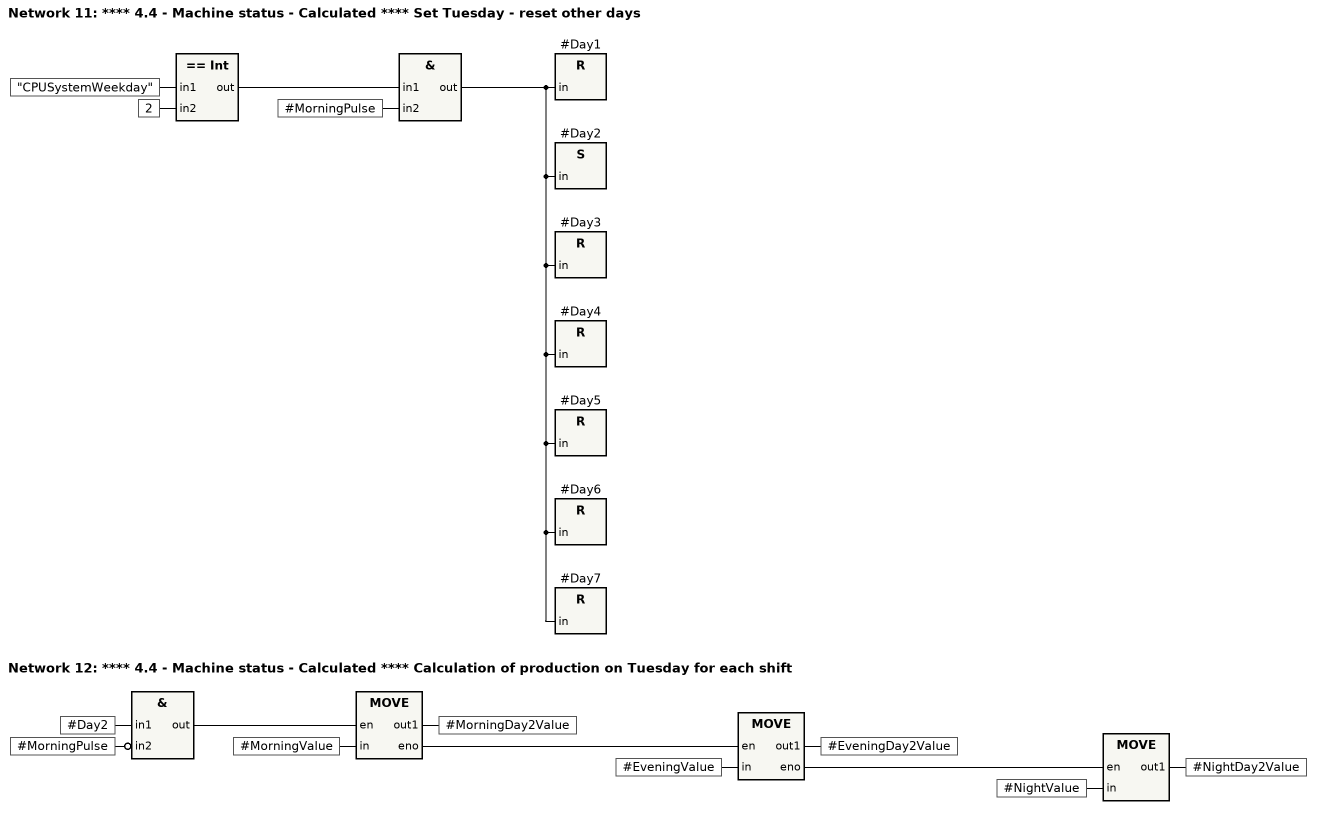
   IF ("CPUSystemWeekday" = 2) AND #MorningPulse THEN
       #Day1 := FALSE;
       #Day2 := TRUE;
       #Day3 := FALSE;
       #Day4 := FALSE;
       #Day5 := FALSE;
       #Day6 := FALSE;
       #Day7 := FALSE;
   END_IF;
END_REGION

REGION Network 12: **** 4.4 - Machine status - Calculated **** Calculation of production on Tuesday for each shift
   // Calculation of production on Tuesday for each shift
   // ENO of a box is taken as its EN; it also drops when the box reports an error
   IF #Day2 AND NOT #MorningPulse THEN
       #MorningDay2Value := #MorningValue;
       #EveningDay2Value := #EveningValue;
       #NightDay2Value := #NightValue;
   END_IF;
END_REGION

NETWORK
TITLE = **** 4.4 - Machine status - Calculated **** Total production on Thuesday
// Total production on Thuesday
      L     #MorningDay2Value;  // amount of bodies on day 2 - Morning shift (Tuesday)
      L     #EveningDay2Value;  // amount of bodies on day 2 - Evening shift (Tuesday)
      +I;
      L     #NightDay2Value;  // amount of bodies on day 2 - Night shift (Tuesday)
      +I;
      T     #Day2Value;  // amount of bodies on day 2 (Tuesday)

REGION Network 14: **** 4.4 - Machine status - Calculated **** Set Wednesday - reset other days
   // Set Wednesday - reset other days
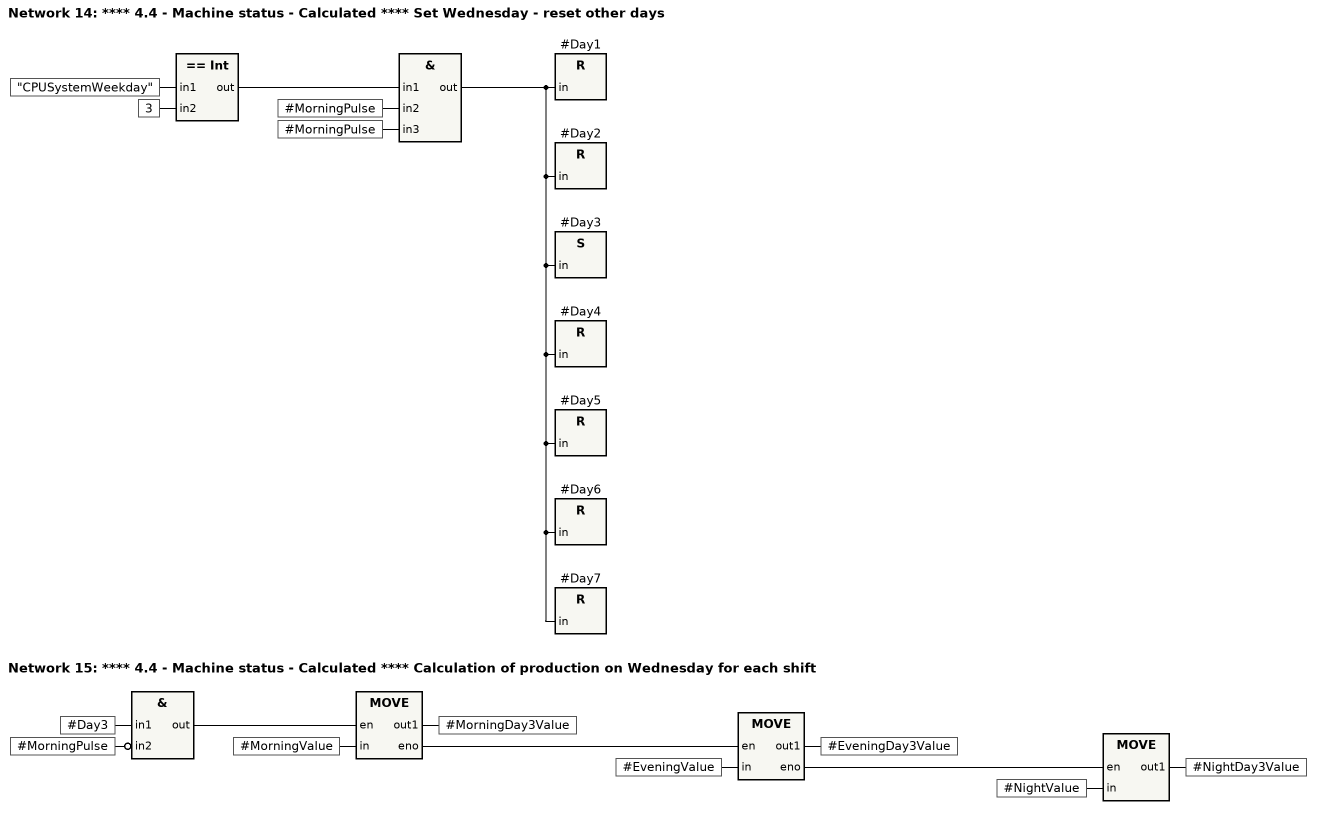
   IF ("CPUSystemWeekday" = 3) AND #MorningPulse AND #MorningPulse THEN
       #Day1 := FALSE;
       #Day2 := FALSE;
       #Day3 := TRUE;
       #Day4 := FALSE;
       #Day5 := FALSE;
       #Day6 := FALSE;
       #Day7 := FALSE;
   END_IF;
END_REGION

REGION Network 15: **** 4.4 - Machine status - Calculated **** Calculation of production on Wednesday for each shift
   // Calculation of production on Wednesday for each shift
   // ENO of a box is taken as its EN; it also drops when the box reports an error
   IF #Day3 AND NOT #MorningPulse THEN
       #MorningDay3Value := #MorningValue;
       #EveningDay3Value := #EveningValue;
       #NightDay3Value := #NightValue;
   END_IF;
END_REGION

NETWORK
TITLE = **** 4.4 - Machine status - Calculated **** Total production on Wednesday
// Total production on Wednesday
      L     #MorningDay3Value;  // amount of bodies on day 3 - Morning shift (Wednesday)
      L     #EveningDay3Value;  // amount of bodies on day 3 - Evening shift (Wednesday)
      +I;
      L     #NightDay3Value;  // amount of bodies on day 3 - Night shift (Wednesday)
      +I;
      T     #Day3Value;  // amount of bodies on day 3 (Wednesday)

REGION Network 17: **** 4.4 - Machine status - Calculated **** Set Thursday - reset other days
   // Set Thursday - reset other days
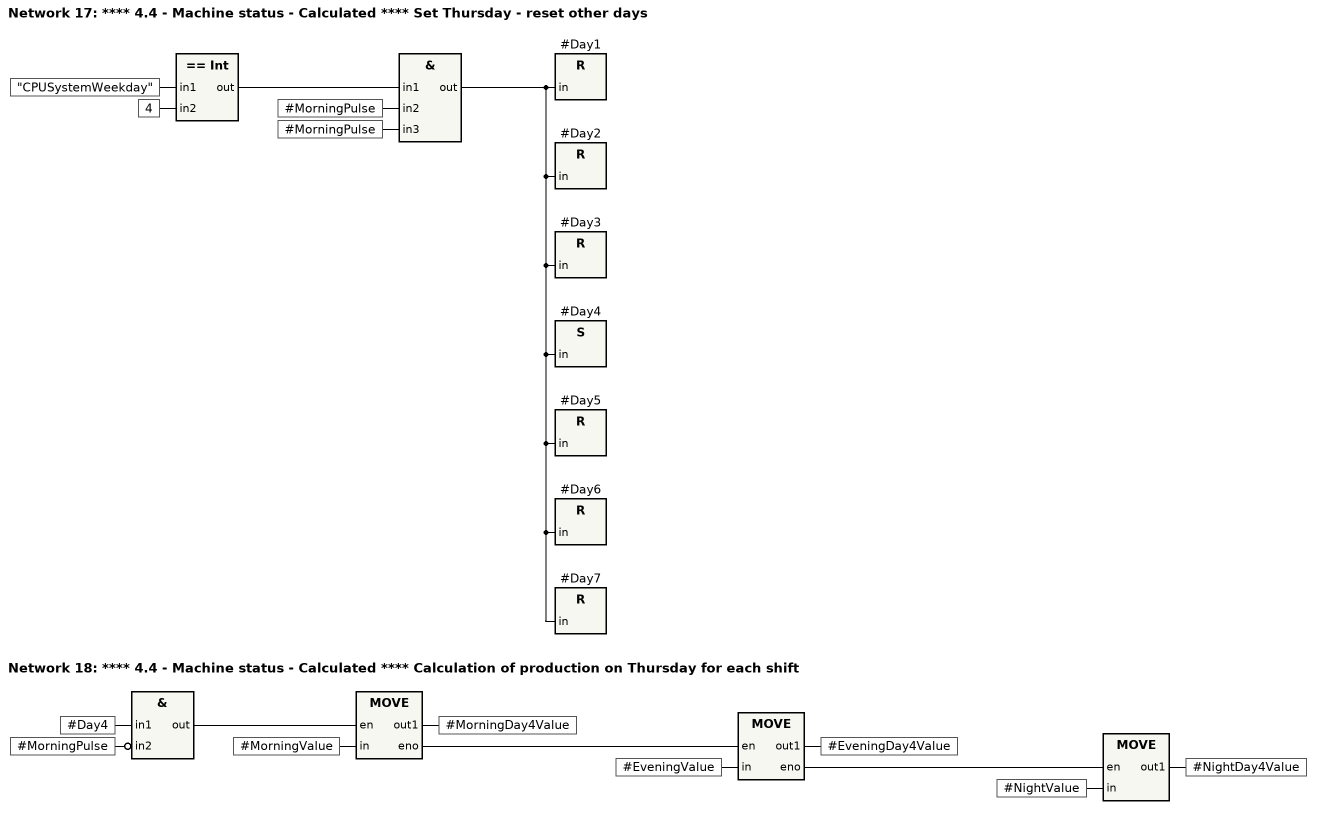
   IF ("CPUSystemWeekday" = 4) AND #MorningPulse AND #MorningPulse THEN
       #Day1 := FALSE;
       #Day2 := FALSE;
       #Day3 := FALSE;
       #Day4 := TRUE;
       #Day5 := FALSE;
       #Day6 := FALSE;
       #Day7 := FALSE;
   END_IF;
END_REGION

REGION Network 18: **** 4.4 - Machine status - Calculated **** Calculation of production on Thursday for each shift
   // Calculation of production on Thursday for each shift
   // ENO of a box is taken as its EN; it also drops when the box reports an error
   IF #Day4 AND NOT #MorningPulse THEN
       #MorningDay4Value := #MorningValue;
       #EveningDay4Value := #EveningValue;
       #NightDay4Value := #NightValue;
   END_IF;
END_REGION

NETWORK
TITLE = **** 4.4 - Machine status - Calculated **** Total production on Thursday
// Total production on Thursday
      L     #MorningDay4Value;  // amount of bodies on day 4 - Morning shift (Thursday)
      L     #EveningDay4Value;  // amount of bodies on day 4 - Evening shift (Thursday)
      +I;
      L     #NightDay4Value;  // amount of bodies on day 4 - Night shift (Thursday)
      +I;
      T     #Day4Value;  // amount of bodies on day 4 (Thursday)

REGION Network 20: **** 4.4 - Machine status - Calculated **** Set Friday - reset other days
   // Set Friday - reset other days
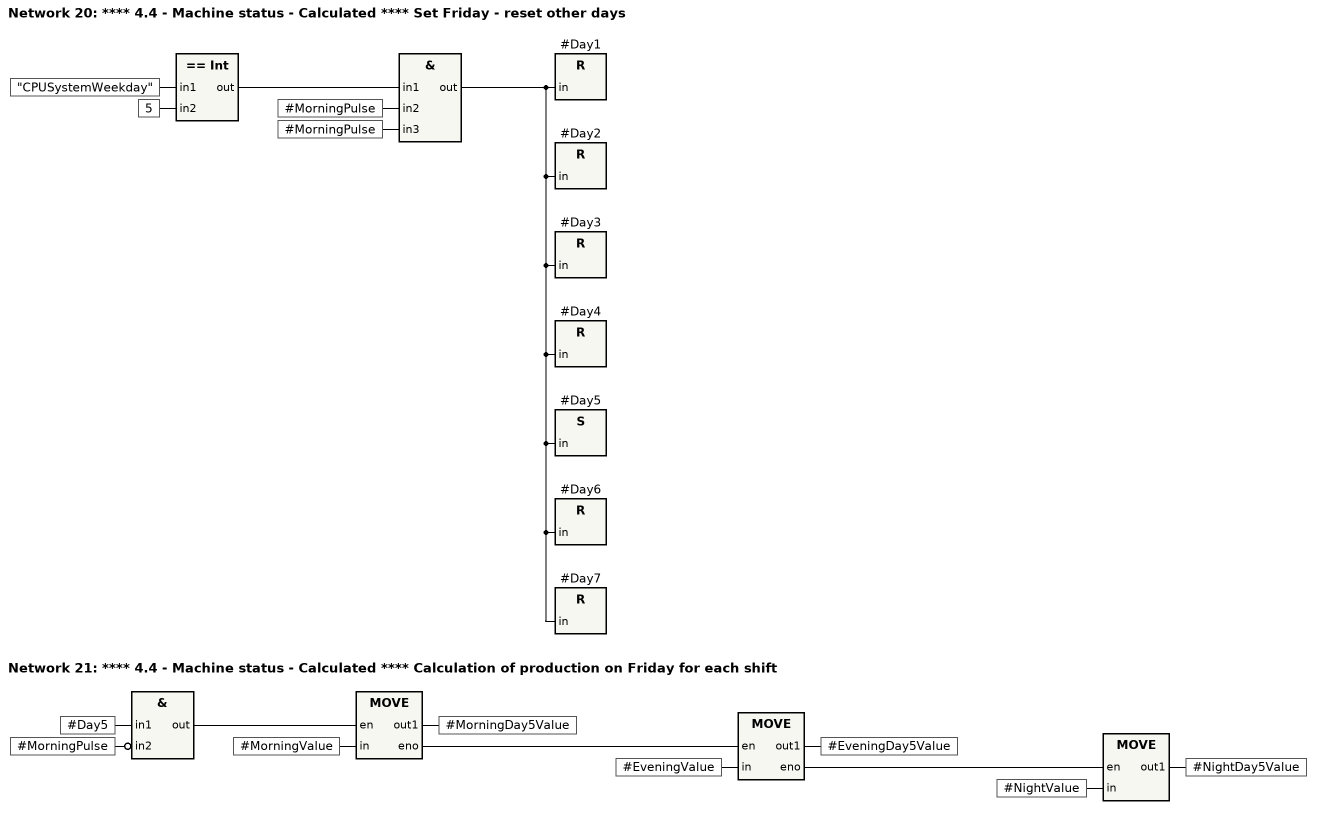
   IF ("CPUSystemWeekday" = 5) AND #MorningPulse AND #MorningPulse THEN
       #Day1 := FALSE;
       #Day2 := FALSE;
       #Day3 := FALSE;
       #Day4 := FALSE;
       #Day5 := TRUE;
       #Day6 := FALSE;
       #Day7 := FALSE;
   END_IF;
END_REGION

REGION Network 21: **** 4.4 - Machine status - Calculated **** Calculation of production on Friday for each shift
   // Calculation of production on Friday for each shift
   // ENO of a box is taken as its EN; it also drops when the box reports an error
   IF #Day5 AND NOT #MorningPulse THEN
       #MorningDay5Value := #MorningValue;
       #EveningDay5Value := #EveningValue;
       #NightDay5Value := #NightValue;
   END_IF;
END_REGION

NETWORK
TITLE = **** 4.4 - Machine status - Calculated **** total production on Friday
// total production on Friday
      L     #MorningDay5Value;  // amount of bodies on day 5 - Morning shift (Friday)
      L     #EveningDay5Value;  // amount of bodies on day 5 - Evening shift (Friday)
      +I;
      L     #NightDay5Value;  // amount of bodies on day 5 - Night shift (Friday)
      +I;
      T     #Day5Value;  // amount of bodies on day 5 (Friday)

REGION Network 23: **** 4.4 - Machine status - Calculated **** Set Saturday - Reset other days
   // Set Saturday - Reset other days
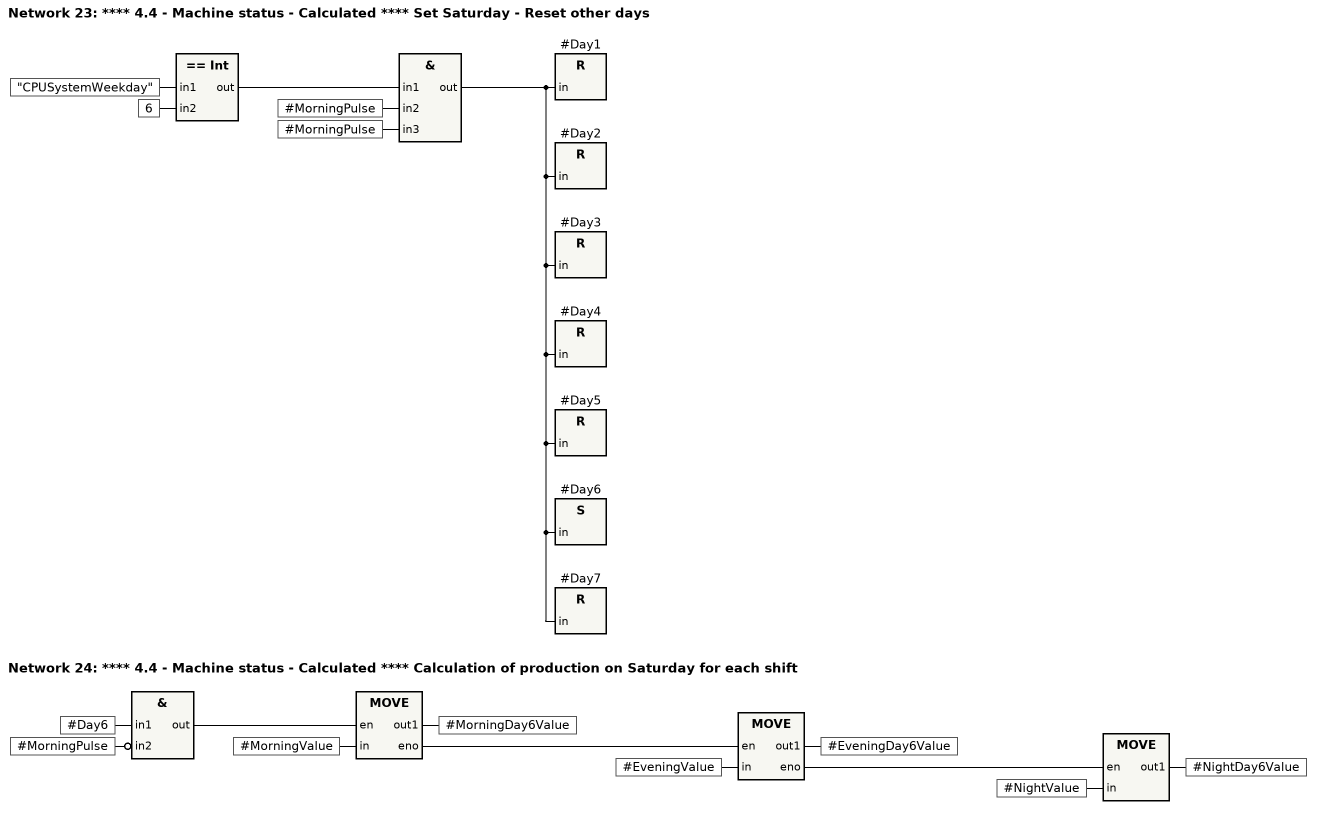
   IF ("CPUSystemWeekday" = 6) AND #MorningPulse AND #MorningPulse THEN
       #Day1 := FALSE;
       #Day2 := FALSE;
       #Day3 := FALSE;
       #Day4 := FALSE;
       #Day5 := FALSE;
       #Day6 := TRUE;
       #Day7 := FALSE;
   END_IF;
END_REGION

REGION Network 24: **** 4.4 - Machine status - Calculated **** Calculation of production on Saturday for each shift
   // Calculation of production on Saturday for each shift
   // ENO of a box is taken as its EN; it also drops when the box reports an error
   IF #Day6 AND NOT #MorningPulse THEN
       #MorningDay6Value := #MorningValue;
       #EveningDay6Value := #EveningValue;
       #NightDay6Value := #NightValue;
   END_IF;
END_REGION

NETWORK
TITLE = **** 4.4 - Machine status - Calculated **** total production on Saturday
// total production on Saturday
      L     #MorningDay6Value;  // amount of bodies on day 6 - Morning shift (Saturday)
      L     #EveningDay6Value;  // amount of bodies on day 6 - Evening shift (Saturday)
      +I;
      L     #NightDay6Value;  // amount of bodies on day 6 - Night shift (Saturday)
      +I;
      T     #Day6Value;  // amount of bodies on day 6 (Saturday)

REGION Network 26: **** 4.4 - Machine status - Calculated **** Set Sunday - Reset other days
   // Set Sunday - Reset other days
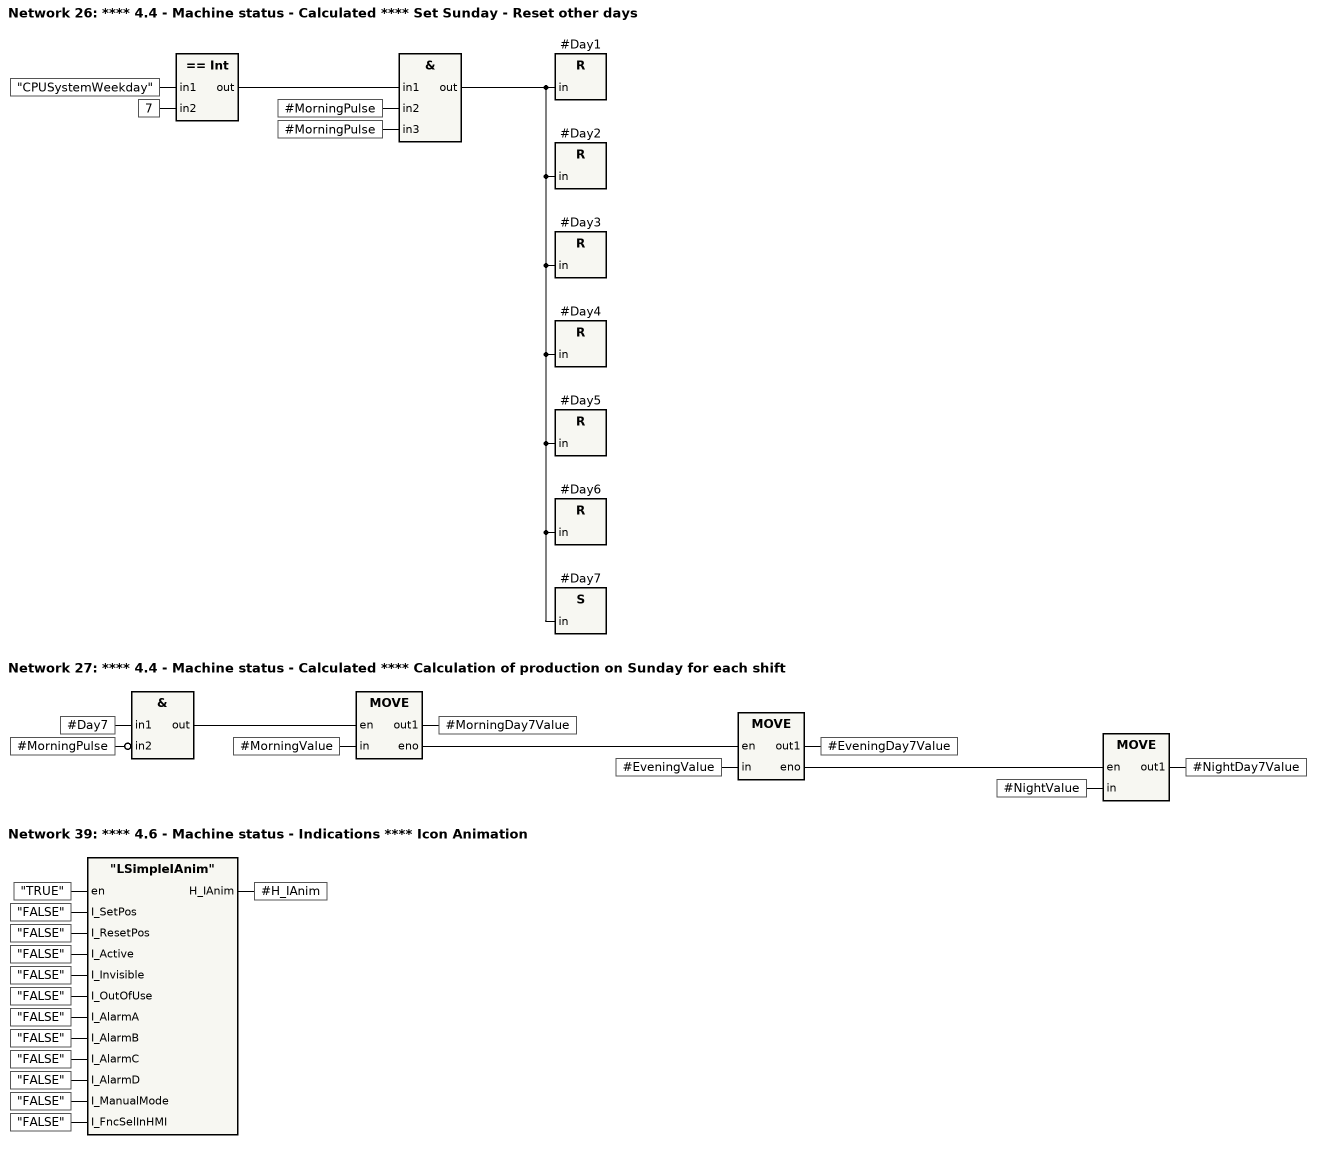
   IF ("CPUSystemWeekday" = 7) AND #MorningPulse AND #MorningPulse THEN
       #Day1 := FALSE;
       #Day2 := FALSE;
       #Day3 := FALSE;
       #Day4 := FALSE;
       #Day5 := FALSE;
       #Day6 := FALSE;
       #Day7 := TRUE;
   END_IF;
END_REGION

REGION Network 27: **** 4.4 - Machine status - Calculated **** Calculation of production on Sunday for each shift
   // Calculation of production on Sunday for each shift
   // ENO of a box is taken as its EN; it also drops when the box reports an error
   IF #Day7 AND NOT #MorningPulse THEN
       #MorningDay7Value := #MorningValue;
       #EveningDay7Value := #EveningValue;
       #NightDay7Value := #NightValue;
   END_IF;
END_REGION

NETWORK
TITLE = **** 4.4 - Machine status - Calculated **** Total production on Sunday
// Total production on Sunday
      L     #MorningDay7Value;  // amount of bodies on day 7 - Morning shift (Sunday)
      L     #EveningDay7Value;  // amount of bodies on day 7 - Evening shift (Sunday)
      +I;
      L     #NightDay7Value;  // amount of bodies on day 7 - Night shift (Sunday)
      +I;
      T     #Day7Value;  // amount of bodies on day 7 (Sunday)

NETWORK
TITLE = **** 4.4 - Machine status - Calculated **** Production value Morning shift
// Production value Morning shift
      A     #Day1;  // Day 1 (Monday)
      JNB   MD1;
      L     #MorningDay1Value;  // amount of bodies on day 1 - Morning shift (Monday)
      T     #H_Out.TotalMorning;  // copy to HMI
MD1:  NOP   0;

      A     #Day2;  // Day 2 (tuesday)
      JNB   MD2;
      L     #MorningDay1Value;  // amount of bodies on day 1 - Morning shift (Monday)
      L     #MorningDay2Value;  // amount of bodies on day 2 - Morning shift (Tuesday)
      T     #H_Out.TotalMorning;  // copy to HMI
MD2:  NOP   0;

      A     #Day3;  // Day 3 (Wednesday)
      JNB   MD3;
      L     #MorningDay1Value;  // amount of bodies on day 1 - Morning shift (Monday)
      L     #MorningDay2Value;  // amount of bodies on day 2 - Morning shift (Tuesday)
      +I;
      L     #MorningDay3Value;  // amount of bodies on day 3 - Morning shift (Wednesday)
      +I;
      T     #H_Out.TotalMorning;  // copy to HMI
MD3:  NOP   0;

      A     #Day4;  // Day 4 (tuesday)
      JNB   MD4;
      L     #MorningDay1Value;  // amount of bodies on day 1 - Morning shift (Monday)
      L     #MorningDay2Value;  // amount of bodies on day 2 - Morning shift (Tuesday)
      +I;
      L     #MorningDay3Value;  // amount of bodies on day 3 - Morning shift (Wednesday)
      +I;
      L     #MorningDay4Value;  // amount of bodies on day 4 - Morning shift (Thursday)
      +I;
      T     #H_Out.TotalMorning;  // copy to HMI
MD4:  NOP   0;

      A     #Day5;  // Day 5 (Friday)
      JNB   MD5;
      L     #MorningDay1Value;  // amount of bodies on day 1 - Morning shift (Monday)
      L     #MorningDay2Value;  // amount of bodies on day 2 - Morning shift (Tuesday)
      +I;
      L     #MorningDay3Value;  // amount of bodies on day 3 - Morning shift (Wednesday)
      +I;
      L     #MorningDay4Value;  // amount of bodies on day 4 - Morning shift (Thursday)
      +I;
      L     #MorningDay5Value;  // amount of bodies on day 5 - Morning shift (Friday)
      +I;
      T     #H_Out.TotalMorning;  // copy to HMI
MD5:  NOP   0;

      A     #Day6;  // Day 6 (Saturday)
      JNB   MD6;
      L     #MorningDay1Value;  // amount of bodies on day 1 - Morning shift (Monday)
      L     #MorningDay2Value;  // amount of bodies on day 2 - Morning shift (Tuesday)
      +I;
      L     #MorningDay3Value;  // amount of bodies on day 3 - Morning shift (Wednesday)
      +I;
      L     #MorningDay4Value;  // amount of bodies on day 4 - Morning shift (Thursday)
      +I;
      L     #MorningDay5Value;  // amount of bodies on day 5 - Morning shift (Friday)
      +I;
      L     #MorningDay6Value;  // amount of bodies on day 6 - Morning shift (Saturday)
      +I;
      T     #H_Out.TotalMorning;  // copy to HMI
MD6:  NOP   0;

      A     #Day7;  // Day 7 (Sunday)
      JNB   MD7;
      L     #MorningDay1Value;  // amount of bodies on day 1 - Morning shift (Monday)
      L     #MorningDay2Value;  // amount of bodies on day 2 - Morning shift (Tuesday)
      +I;
      L     #MorningDay3Value;  // amount of bodies on day 3 - Morning shift (Wednesday)
      +I;
      L     #MorningDay4Value;  // amount of bodies on day 4 - Morning shift (Thursday)
      +I;
      L     #MorningDay5Value;  // amount of bodies on day 5 - Morning shift (Friday)
      +I;
      L     #MorningDay6Value;  // amount of bodies on day 6 - Morning shift (Saturday)
      +I;
      L     #MorningDay7Value;  // amount of bodies on day 7 - Morning shift (Sunday)
      +I;
      T     #H_Out.TotalMorning;  // copy to HMI
MD7:  NOP   0;


NETWORK
TITLE = **** 4.4 - Machine status - Calculated **** Production value Evening shift
// Production value Evening shift
      A     #Day1;  // Day 1 (Monday)
      JNB   ED1;
      L     #EveningDay1Value;  // amount of bodies on day 1 - Evening shift (Monday)
      T     #H_Out.TotalEvening;  // copy to HMI
ED1:  NOP   0;

      A     #Day2;  // Day 2 (tuesday)
      JNB   ED2;
      L     #EveningDay1Value;  // amount of bodies on day 1 - Evening shift (Monday)
      L     #EveningDay2Value;  // amount of bodies on day 2 - Evening shift (Tuesday)
      T     #H_Out.TotalEvening;  // copy to HMI
ED2:  NOP   0;

      A     #Day3;  // Day 3 (Wednesday)
      JNB   ED3;
      L     #EveningDay1Value;  // amount of bodies on day 1 - Evening shift (Monday)
      L     #EveningDay2Value;  // amount of bodies on day 2 - Evening shift (Tuesday)
      +I;
      L     #EveningDay3Value;  // amount of bodies on day 3 - Evening shift (Wednesday)
      +I;
      T     #H_Out.TotalEvening;  // copy to HMI
ED3:  NOP   0;

      A     #Day4;  // Day 4 (tuesday)
      JNB   ED4;
      L     #EveningDay1Value;  // amount of bodies on day 1 - Evening shift (Monday)
      L     #EveningDay2Value;  // amount of bodies on day 2 - Evening shift (Tuesday)
      +I;
      L     #EveningDay3Value;  // amount of bodies on day 3 - Evening shift (Wednesday)
      +I;
      L     #EveningDay4Value;  // amount of bodies on day 4 - Evening shift (Thursday)
      +I;
      T     #H_Out.TotalEvening;  // copy to HMI
ED4:  NOP   0;

      A     #Day5;  // Day 5 (Friday)
      JNB   ED5;
      L     #EveningDay1Value;  // amount of bodies on day 1 - Evening shift (Monday)
      L     #EveningDay2Value;  // amount of bodies on day 2 - Evening shift (Tuesday)
      +I;
      L     #EveningDay3Value;  // amount of bodies on day 3 - Evening shift (Wednesday)
      +I;
      L     #EveningDay4Value;  // amount of bodies on day 4 - Evening shift (Thursday)
      +I;
      L     #EveningDay5Value;  // amount of bodies on day 5 - Evening shift (Friday)
      +I;
      T     #H_Out.TotalEvening;  // copy to HMI
ED5:  NOP   0;

